LIN {X 0,Y 514.264,Z 1274.266,A -85,B 0,C 180,E1 4933.156,E2 4933.156} C_VEL
LIN {X 0,Y 513.464,Z 1291.981,A -85,B 0,C 180,E1 4937.266,E2 4937.266} C_VEL
LIN {X 0,Y 513.172,Z 1303.726,A -85,B 0,C 180,E1 4941.123,E2 4941.123} C_VEL
LIN {X 0,Y 512.967,Z 1310.956,A -85,B 0,C 180,E1 4944.936,E2 4944.936} C_VEL
LIN {X 0,Y 512.995,Z 1314.088,A -85,B 0,C 180,E1 4948.314,E2 4948.314} C_VEL
LIN {X 0,Y 513.103,Z 1314.089,A -85,B 0,C 180,E1 4951.685,E2 4951.685} C_VEL
LIN {X 0,Y 513.097,Z 1309.756,A -85,B 0,C 180,E1 4955.908,E2 4955.908} C_VEL
LIN {X 0,Y 513.202,Z 1300.306,A -85,B 0,C 180,E1 4960.161,E2 4960.161} C_VEL
LIN {X 0,Y 513.734,Z 1286.168,A -85,B 0,C 180,E1 4964.239,E2 4964.239} C_VEL
LIN {X 0,Y 514.771,Z 1266.36,A -85,B 0,C 180,E1 4968.328,E2 4968.328} C_VEL
LIN {X 0,Y 516.526,Z 1240.321,A -85,B 0,C 180,E1 4972.32,E2 4972.32} C_VEL
LIN {X 0,Y 518.823,Z 1209.462,A -85,B 0,C 180,E1 4975.866,E2 4975.866} C_VEL
LIN {X 0,Y 521.361,Z 1175.943,A -85,B 0,C 180,E1 4978.762,E2 4978.762} C_VEL
LIN {X 0,Y 523.842,Z 1140.515,A -85,B 0,C 180,E1 4981.019,E2 4981.019} C_VEL
LIN {X 0,Y 525.891,Z 1102.955,A -85,B 0,C 180,E1 4982.687,E2 4982.687} C_VEL
LIN {X 0,Y 527.428,Z 1065.762,A -85,B 0,C 180,E1 4983.695,E2 4983.695} C_VEL
LIN {X 0,Y 527.288,Z 1021.079,A -85,B 0,C 180,E1 4984.459,E2 4984.459} C_VEL
LIN {X 0,Y 512.361,Z 989.03,A -85,B 0,C 180,E1 4986.22,E2 4986.22} C_VEL
LIN {X 0,Y 512.298,Z 989.03,A -85,B 0,C 180,E1 4990.392,E2 4990.392} C_VEL
LIN {X 0,Y 512.249,Z 989.03,A -85,B 0,C 180,E1 4997.35,E2 4997.35} C_VEL
LIN {X 0,Y 512.299,Z 989.03,A -85,B 0,C 180,E1 5002.683,E2 5002.683} C_VEL
LIN {X 0,Y 512.294,Z 989.03,A -85,B 0,C 180,E1 5008.673,E2 5008.673} C_VEL
LIN {X 0,Y 512.37,Z 989.03,A -85,B 0,C 180,E1 5013.784,E2 5013.784} C_VEL
LIN {X 0,Y 512.546,Z 989.03,A -85,B 0,C 180,E1 5019.312,E2 5019.312} C_VEL
LIN {X 0,Y 512.454,Z 989.03,A -85,B 0,C 180,E1 5024.632,E2 5024.632} C_VEL
LIN {X 0,Y 512.627,Z 989.03,A -85,B 0,C 180,E1 5029.827,E2 5029.827} C_VEL
LIN {X 0,Y 512.838,Z 989.03,A -85,B 0,C 180,E1 5034.936,E2 5034.936} C_VEL
LIN {X 0,Y 512.854,Z 989.03,A -85,B 0,C 180,E1 5040,E2 5040} C_VEL
LIN {X 0,Y 512.807,Z 989.03,A -85,B 0,C 180,E1 5045.064,E2 5045.064} C_VEL
LIN {X 0,Y 512.702,Z 989.03,A -85,B 0,C 180,E1 5050.171,E2 5050.171} C_VEL
LIN {X 0,Y 512.597,Z 989.03,A -85,B 0,C 180,E1 5055.363,E2 5055.363} C_VEL
LIN {X 0,Y 512.537,Z 989.03,A -85,B 0,C 180,E1 5060.689,E2 5060.689} C_VEL
LIN {X 0,Y 512.336,Z 989.03,A -85,B 0,C 180,E1 5066.218,E2 5066.218} C_VEL
LIN {X 0,Y 512.295,Z 989.03,A -85,B 0,C 180,E1 5072.018,E2 5072.018} C_VEL
LIN {X 0,Y 512.168,Z 989.03,A -85,B 0,C 180,E1 5078.221,E2 5078.221} C_VEL
LIN {X 0,Y 512.21,Z 989.03,A -85,B 0,C 180,E1 5084.994,E2 5084.994} C_VEL
LIN {X 0,Y 512.302,Z 989.03,A -85,B 0,C 180,E1 5089.979,E2 5089.979} C_VEL
LIN {X 0,Y 512.239,Z 989.03,A -85,B 0,C 180,E1 5095.964,E2 5095.964} C_VEL
LIN {X 0,Y 512.363,Z 989.065,A -85,B 0,C 180,E1 5098.077,E2 5098.077} C_VEL
LIN {X 0,Y 521.604,Z 1021.148,A -85,B 0,C 180,E1 5100.836,E2 5100.836} C_VEL
LIN {X 0,Y 519.15,Z 1055.325,A -85,B 0,C 180,E1 5103.688,E2 5103.688} C_VEL
LIN {X 0,Y 516.857,Z 1085.604,A -85,B 0,C 180,E1 5107.034,E2 5107.034} C_VEL
LIN {X 0,Y 515.067,Z 1111.372,A -85,B 0,C 180,E1 5110.771,E2 5110.771} C_VEL
LIN {X 0,Y 513.907,Z 1131.701,A -85,B 0,C 180,E1 5114.677,E2 5114.677} C_VEL
LIN {X 0,Y 513.347,Z 1147.878,A -85,B 0,C 180,E1 5118.985,E2 5118.985} C_VEL
LIN {X 0,Y 513.104,Z 1158.306,A -85,B 0,C 180,E1 5123.245,E2 5123.245} C_VEL
LIN {X 0,Y 512.989,Z 1162.956,A -85,B 0,C 180,E1 5126.628,E2 5126.628} C_VEL
LIN {X 0,Y 513.004,Z 1164.497,A -85,B 0,C 180,E1 5130.001,E2 5130.001} C_VEL
LIN {X 0,Y 512.994,Z 1162.865,A -85,B 0,C 180,E1 5133.373,E2 5133.373} C_VEL
LIN {X 0,Y 513.065,Z 1156.495,A -85,B 0,C 180,E1 5137.606,E2 5137.606} C_VEL
LIN {X 0,Y 513.404,Z 1144.882,A -85,B 0,C 180,E1 5141.874,E2 5141.874} C_VEL
LIN {X 0,Y 514.188,Z 1127.29,A -85,B 0,C 180,E1 5146.189,E2 5146.189} C_VEL
LIN {X 0,Y 515.459,Z 1105.361,A -85,B 0,C 180,E1 5150.113,E2 5150.113} C_VEL
LIN {X 0,Y 517.484,Z 1077.478,A -85,B 0,C 180,E1 5153.867,E2 5153.867} C_VEL
LIN {X 0,Y 519.839,Z 1045.937,A -85,B 0,C 180,E1 5157.09,E2 5157.09} C_VEL
LIN {X 0,Y 521.275,Z 1018.437,A -85,B 0,C 180,E1 5159.305,E2 5159.305} C_VEL
LIN {X 0,Y 512.342,Z 989.03,A -85,B 0,C 180,E1 5161.88,E2 5161.88} C_VEL
LIN {X 0,Y 512.182,Z 989.03,A -85,B 0,C 180,E1 5168.223,E2 5168.223} C_VEL
LIN {X 0,Y 512.218,Z 989.03,A -85,B 0,C 180,E1 5175.007,E2 5175.007} C_VEL
LIN {X 0,Y 512.311,Z 989.03,A -85,B 0,C 180,E1 5179.982,E2 5179.982} C_VEL
LIN {X 0,Y 512.229,Z 989.03,A -85,B 0,C 180,E1 5185.964,E2 5185.964} C_VEL
LIN {X 0,Y 512.354,Z 989.03,A -85,B 0,C 180,E1 5192.078,E2 5192.078} C_VEL
LIN {X 0,Y 512.457,Z 989.03,A -85,B 0,C 180,E1 5197.494,E2 5197.494} C_VEL
LIN {X 0,Y 512.639,Z 989.03,A -85,B 0,C 180,E1 5202.882,E2 5202.882} C_VEL
LIN {X 0,Y 512.635,Z 989.03,A -85,B 0,C 180,E1 5209.828,E2 5209.828} C_VEL
LIN {X 0,Y 512.85,Z 989.03,A -85,B 0,C 180,E1 5214.936,E2 5214.936} C_VEL
LIN {X 0,Y 512.911,Z 989.03,A -85,B 0,C 180,E1 5220,E2 5220} C_VEL
LIN {X 0,Y 512.831,Z 989.03,A -85,B 0,C 180,E1 5225.064,E2 5225.064} C_VEL
LIN {X 0,Y 512.709,Z 989.03,A -85,B 0,C 180,E1 5230.171,E2 5230.171} C_VEL
LIN {X 0,Y 512.61,Z 989.03,A -85,B 0,C 180,E1 5235.363,E2 5235.363} C_VEL
LIN {X 0,Y 512.534,Z 989.03,A -85,B 0,C 180,E1 5240.689,E2 5240.689} C_VEL
LIN {X 0,Y 512.344,Z 989.03,A -85,B 0,C 180,E1 5246.217,E2 5246.217} C_VEL
LIN {X 0,Y 512.44,Z 989.03,A -85,B 0,C 180,E1 5252.008,E2 5252.008} C_VEL
LIN {X 0,Y 512.33,Z 989.03,A -85,B 0,C 180,E1 5258.061,E2 5258.061} C_VEL
LIN {X 0,Y 509.805,Z 989.03,A -85,B 0,C 180,E1 5259.49,E2 5259.49} C_VEL
LIN {X 0,Y 504.194,Z 989.03,A -85,B 0,C 180,E1 5261.878,E2 5261.878} C_VEL
LIN {X 0,Y 504.274,Z 989.03,A -85,B 0,C 180,E1 5268.424,E2 5268.424} C_VEL
LIN {X 0,Y 504.544,Z 989.315,A -85,B 0,C 180,E1 5273.26,E2 5273.26} C_VEL
LIN {X 0,Y 521.241,Z 1024.493,A -85,B 0,C 180,E1 5275.14,E2 5275.14} C_VEL
LIN {X 0,Y 520.227,Z 1081.386,A -85,B 0,C 180,E1 5276.169,E2 5276.169} C_VEL
LIN {X 0,Y 518.352,Z 1120.193,A -85,B 0,C 180,E1 5277.525,E2 5277.525} C_VEL
LIN {X 0,Y 515.742,Z 1157.972,A -85,B 0,C 180,E1 5279.553,E2 5279.553} C_VEL
LIN {X 0,Y 512.859,Z 1193.587,A -85,B 0,C 180,E1 5282.243,E2 5282.243} C_VEL
LIN {X 0,Y 510.276,Z 1224.521,A -85,B 0,C 180,E1 5285.369,E2 5285.369} C_VEL
LIN {X 0,Y 508.165,Z 1251.245,A -85,B 0,C 180,E1 5288.896,E2 5288.896} C_VEL
LIN {X 0,Y 506.553,Z 1274.264,A -85,B 0,C 180,E1 5292.891,E2 5292.891} C_VEL
LIN {X 0,Y 505.643,Z 1291.982,A -85,B 0,C 180,E1 5297.066,E2 5297.066} C_VEL
LIN {X 0,Y 505.264,Z 1304.676,A -85,B 0,C 180,E1 5301.411,E2 5301.411} C_VEL
LIN {X 0,Y 505.074,Z 1310.957,A -85,B 0,C 180,E1 5304.857,E2 5304.857} C_VEL
LIN {X 0,Y 505.093,Z 1314.088,A -85,B 0,C 180,E1 5308.287,E2 5308.287} C_VEL
LIN {X 0,Y 505.196,Z 1314.089,A -85,B 0,C 180,E1 5311.711,E2 5311.711} C_VEL
LIN {X 0,Y 505.205,Z 1309.756,A -85,B 0,C 180,E1 5316,E2 5316} C_VEL
LIN {X 0,Y 505.319,Z 1300.306,A -85,B 0,C 180,E1 5320.321,E2 5320.321} C_VEL
LIN {X 0,Y 505.986,Z 1285.076,A -85,B 0,C 180,E1 5324.738,E2 5324.738} C_VEL
LIN {X 0,Y 507.27,Z 1263.662,A -85,B 0,C 180,E1 5329.1,E2 5329.1} C_VEL
LIN {X 0,Y 509.094,Z 1238.474,A -85,B 0,C 180,E1 5332.912,E2 5332.912} C_VEL
LIN {X 0,Y 511.597,Z 1208.319,A -85,B 0,C 180,E1 5336.377,E2 5336.377} C_VEL
LIN {X 0,Y 514.358,Z 1175.174,A -85,B 0,C 180,E1 5339.252,E2 5339.252} C_VEL
LIN {X 0,Y 517.035,Z 1139.614,A -85,B 0,C 180,E1 5341.525,E2 5341.525} C_VEL
LIN {X 0,Y 519.276,Z 1101.697,A -85,B 0,C 180,E1 5343.205,E2 5343.205} C_VEL
LIN {X 0,Y 520.948,Z 1063.021,A -85,B 0,C 180,E1 5344.225,E2 5344.225} C_VEL
LIN {X 0,Y 520.741,Z 1023.716,A -85,B 0,C 180,E1 5344.911,E2 5344.911} C_VEL
LIN {X 0,Y 504.482,Z 989.03,A -85,B 0,C 180,E1 5346.818,E2 5346.818} C_VEL
LIN {X 0,Y 504.197,Z 989.03,A -85,B 0,C 180,E1 5353.5,E2 5353.5} C_VEL
LIN {X 0,Y 504.287,Z 989.03,A -85,B 0,C 180,E1 5358.83,E2 5358.83} C_VEL
LIN {X 0,Y 504.4,Z 989.03,A -85,B 0,C 180,E1 5363.876,E2 5363.876} C_VEL
LIN {X 0,Y 504.349,Z 989.03,A -85,B 0,C 180,E1 5370.189,E2 5370.189} C_VEL
LIN {X 0,Y 504.437,Z 989.03,A -85,B 0,C 180,E1 5375.242,E2 5375.242} C_VEL
LIN {X 0,Y 504.662,Z 989.03,A -85,B 0,C 180,E1 5380.798,E2 5380.798} C_VEL
LIN {X 0,Y 504.474,Z 989.03,A -85,B 0,C 180,E1 5386.155,E2 5386.155} C_VEL
LIN {X 0,Y 504.709,Z 989.03,A -85,B 0,C 180,E1 5391.403,E2 5391.403} C_VEL
LIN {X 0,Y 504.868,Z 989.03,A -85,B 0,C 180,E1 5396.573,E2 5396.573} C_VEL
LIN {X 0,Y 504.878,Z 989.03,A -85,B 0,C 180,E1 5401.713,E2 5401.713} C_VEL
LIN {X 0,Y 504.801,Z 989.03,A -85,B 0,C 180,E1 5406.867,E2 5406.867} C_VEL
LIN {X 0,Y 504.723,Z 989.03,A -85,B 0,C 180,E1 5412.08,E2 5412.08} C_VEL
LIN {X 0,Y 504.674,Z 989.03,A -85,B 0,C 180,E1 5417.397,E2 5417.397} C_VEL
LIN {X 0,Y 504.538,Z 989.03,A -85,B 0,C 180,E1 5422.88,E2 5422.88} C_VEL
LIN {X 0,Y 504.372,Z 989.03,A -85,B 0,C 180,E1 5428.599,E2 5428.599} C_VEL
LIN {X 0,Y 504.304,Z 989.03,A -85,B 0,C 180,E1 5434.646,E2 5434.646} C_VEL
LIN {X 0,Y 504.179,Z 989.03,A -85,B 0,C 180,E1 5441.18,E2 5441.18} C_VEL
LIN {X 0,Y 504.236,Z 989.03,A -85,B 0,C 180,E1 5446.504,E2 5446.504} C_VEL
LIN {X 0,Y 504.388,Z 989.03,A -85,B 0,C 180,E1 5453.249,E2 5453.249} C_VEL
LIN {X 0,Y 504.392,Z 989.133,A -85,B 0,C 180,E1 5457.512,E2 5457.512} C_VEL
LIN {X 0,Y 514.407,Z 1023.254,A -85,B 0,C 180,E1 5460.555,E2 5460.555} C_VEL
LIN {X 0,Y 511.797,Z 1056.465,A -85,B 0,C 180,E1 5463.398,E2 5463.398} C_VEL
LIN {X 0,Y 509.247,Z 1087.005,A -85,B 0,C 180,E1 5466.856,E2 5466.856} C_VEL
LIN {X 0,Y 507.312,Z 1112.759,A -85,B 0,C 180,E1 5470.702,E2 5470.702} C_VEL
LIN {X 0,Y 506.058,Z 1134.079,A -85,B 0,C 180,E1 5474.976,E2 5474.976} C_VEL
LIN {X 0,Y 505.494,Z 1150.423,A -85,B 0,C 180,E1 5479.682,E2 5479.682} C_VEL
LIN {X 0,Y 505.204,Z 1159.82,A -85,B 0,C 180,E1 5484,E2 5484} C_VEL
LIN {X 0,Y 505.088,Z 1164.116,A -85,B 0,C 180,E1 5488.289,E2 5488.289} C_VEL
LIN {X 0,Y 505.203,Z 1164.062,A -85,B 0,C 180,E1 5491.712,E2 5491.712} C_VEL
LIN {X 0,Y 505.158,Z 1159.685,A -85,B 0,C 180,E1 5496.002,E2 5496.002} C_VEL
LIN {X 0,Y 505.36,Z 1150.185,A -85,B 0,C 180,E1 5500.322,E2 5500.322} C_VEL
LIN {X 0,Y 505.989,Z 1134.907,A -85,B 0,C 180,E1 5504.736,E2 5504.736} C_VEL
LIN {X 0,Y 507.272,Z 1113.393,A -85,B 0,C 180,E1 5509.101,E2 5509.101} C_VEL
LIN {X 0,Y 509.165,Z 1088.092,A -85,B 0,C 180,E1 5512.914,E2 5512.914} C_VEL
LIN {X 0,Y 511.655,Z 1057.868,A -85,B 0,C 180,E1 5516.375,E2 5516.375} C_VEL
LIN {X 0,Y 514.45,Z 1024.571,A -85,B 0,C 180,E1 5519.249,E2 5519.249} C_VEL
LIN {X 0,Y 505.519,Z 992.998,A -85,B 0,C 180,E1 5522.083,E2 5522.083} C_VEL
LIN {X 0,Y 504.383,Z 989.03,A -85,B 0,C 180,E1 5522.459,E2 5522.459} C_VEL
LIN {X 0,Y 504.236,Z 989.03,A -85,B 0,C 180,E1 5528.937,E2 5528.937} C_VEL
LIN {X 0,Y 504.223,Z 989.03,A -85,B 0,C 180,E1 5534.092,E2 5534.092} C_VEL
LIN {X 0,Y 504.302,Z 989.03,A -85,B 0,C 180,E1 5538.832,E2 5538.832} C_VEL
LIN {X 0,Y 504.407,Z 989.03,A -85,B 0,C 180,E1 5543.877,E2 5543.877} C_VEL
LIN {X 0,Y 504.355,Z 989.03,A -85,B 0,C 180,E1 5550.19,E2 5550.19} C_VEL
LIN {X 0,Y 504.444,Z 989.03,A -85,B 0,C 180,E1 5555.242,E2 5555.242} C_VEL
LIN {X 0,Y 504.681,Z 989.03,A -85,B 0,C 180,E1 5560.799,E2 5560.799} C_VEL
LIN {X 0,Y 504.485,Z 989.03,A -85,B 0,C 180,E1 5566.156,E2 5566.156} C_VEL
LIN {X 0,Y 504.737,Z 989.03,A -85,B 0,C 180,E1 5571.403,E2 5571.403} C_VEL
LIN {X 0,Y 504.877,Z 989.03,A -85,B 0,C 180,E1 5576.573,E2 5576.573} C_VEL
LIN {X 0,Y 504.848,Z 989.03,A -85,B 0,C 180,E1 5581.713,E2 5581.713} C_VEL
LIN {X 0,Y 504.81,Z 989.03,A -85,B 0,C 180,E1 5586.867,E2 5586.867} C_VEL
LIN {X 0,Y 504.734,Z 989.03,A -85,B 0,C 180,E1 5592.08,E2 5592.08} C_VEL
LIN {X 0,Y 504.658,Z 989.03,A -85,B 0,C 180,E1 5597.398,E2 5597.398} C_VEL
LIN {X 0,Y 504.506,Z 989.03,A -85,B 0,C 180,E1 5602.881,E2 5602.881} C_VEL
LIN {X 0,Y 504.406,Z 989.03,A -85,B 0,C 180,E1 5608.597,E2 5608.597} C_VEL
LIN {X 0,Y 504.476,Z 989.03,A -85,B 0,C 180,E1 5614.633,E2 5614.633} C_VEL
LIN {X 0,Y 504.264,Z 989.03,A -85,B 0,C 180,E1 5621.172,E2 5621.172} C_VEL
LIN {X 0,Y 504.194,Z 989.03,A -85,B 0,C 180,E1 5621.878,E2 5621.878} C_VEL
LIN {X 0,Y 500.197,Z 989.03,A -85,B 0,C 180,E1 5623.826,E2 5623.826} C_VEL
LIN {X 0,Y 496.264,Z 989.03,A -85,B 0,C 180,E1 5625.804,E2 5625.804} C_VEL
LIN {X 0,Y 496.596,Z 989.03,A -85,B 0,C 180,E1 5632.573,E2 5632.573} C_VEL
LIN {X 0,Y 514.658,Z 1027.323,A -85,B 0,C 180,E1 5634.689,E2 5634.689} C_VEL
LIN {X 0,Y 513.661,Z 1081.286,A -85,B 0,C 180,E1 5635.675,E2 5635.675} C_VEL
LIN {X 0,Y 511.623,Z 1120.474,A -85,B 0,C 180,E1 5637.059,E2 5637.059} C_VEL
LIN {X 0,Y 508.83,Z 1157.545,A -85,B 0,C 180,E1 5639.064,E2 5639.064} C_VEL
LIN {X 0,Y 505.715,Z 1193.156,A -85,B 0,C 180,E1 5641.775,E2 5641.775} C_VEL
LIN {X 0,Y 502.879,Z 1224.715,A -85,B 0,C 180,E1 5645.006,E2 5645.006} C_VEL
LIN {X 0,Y 500.454,Z 1252.697,A -85,B 0,C 180,E1 5648.786,E2 5648.786} C_VEL
LIN {X 0,Y 498.725,Z 1275.344,A -85,B 0,C 180,E1 5652.841,E2 5652.841} C_VEL
LIN {X 0,Y 497.812,Z 1291.982,A -85,B 0,C 180,E1 5656.858,E2 5656.858} C_VEL
LIN {X 0,Y 497.388,Z 1304.676,A -85,B 0,C 180,E1 5661.274,E2 5661.274} C_VEL
LIN {X 0,Y 497.182,Z 1310.957,A -85,B 0,C 180,E1 5664.775,E2 5664.775} C_VEL
LIN {X 0,Y 497.214,Z 1314.088,A -85,B 0,C 180,E1 5668.26,E2 5668.26} C_VEL
LIN {X 0,Y 497.291,Z 1314.089,A -85,B 0,C 180,E1 5671.738,E2 5671.738} C_VEL
LIN {X 0,Y 497.327,Z 1309.755,A -85,B 0,C 180,E1 5676.096,E2 5676.096} C_VEL
LIN {X 0,Y 497.438,Z 1300.306,A -85,B 0,C 180,E1 5680.486,E2 5680.486} C_VEL
LIN {X 0,Y 498.235,Z 1284.679,A -85,B 0,C 180,E1 5685.075,E2 5685.075} C_VEL
LIN {X 0,Y 499.604,Z 1263.661,A -85,B 0,C 180,E1 5689.404,E2 5689.404} C_VEL
LIN {X 0,Y 501.633,Z 1238.473,A -85,B 0,C 180,E1 5693.273,E2 5693.273} C_VEL
LIN {X 0,Y 504.345,Z 1208.416,A -85,B 0,C 180,E1 5696.776,E2 5696.776} C_VEL
LIN {X 0,Y 507.368,Z 1174.406,A -85,B 0,C 180,E1 5699.756,E2 5699.756} C_VEL
LIN {X 0,Y 510.363,Z 1137.859,A -85,B 0,C 180,E1 5702.089,E2 5702.089} C_VEL
LIN {X 0,Y 512.762,Z 1099.707,A -85,B 0,C 180,E1 5703.759,E2 5703.759} C_VEL
LIN {X 0,Y 514.393,Z 1061.693,A -85,B 0,C 180,E1 5704.742,E2 5704.742} C_VEL
LIN {X 0,Y 514.105,Z 1026.127,A -85,B 0,C 180,E1 5705.372,E2 5705.372} C_VEL
LIN {X 0,Y 496.553,Z 989.03,A -85,B 0,C 180,E1 5707.429,E2 5707.429} C_VEL
LIN {X 0,Y 496.322,Z 989.03,A -85,B 0,C 180,E1 5714.369,E2 5714.369} C_VEL
LIN {X 0,Y 496.387,Z 989.03,A -85,B 0,C 180,E1 5720.33,E2 5720.33} C_VEL
LIN {X 0,Y 496.374,Z 989.03,A -85,B 0,C 180,E1 5726.826,E2 5726.826} C_VEL
LIN {X 0,Y 496.475,Z 989.03,A -85,B 0,C 180,E1 5732.877,E2 5732.877} C_VEL
LIN {X 0,Y 496.659,Z 989.03,A -85,B 0,C 180,E1 5738.618,E2 5738.618} C_VEL
LIN {X 0,Y 496.666,Z 989.03,A -85,B 0,C 180,E1 5744.131,E2 5744.131} C_VEL
LIN {X 0,Y 496.773,Z 989.03,A -85,B 0,C 180,E1 5749.499,E2 5749.499} C_VEL
LIN {X 0,Y 497.027,Z 989.03,A -85,B 0,C 180,E1 5754.774,E2 5754.774} C_VEL
LIN {X 0,Y 497.061,Z 989.03,A -85,B 0,C 180,E1 5760,E2 5760} C_VEL
LIN {X 0,Y 496.993,Z 989.03,A -85,B 0,C 180,E1 5765.226,E2 5765.226} C_VEL
LIN {X 0,Y 496.864,Z 989.03,A -85,B 0,C 180,E1 5770.499,E2 5770.499} C_VEL
LIN {X 0,Y 496.754,Z 989.03,A -85,B 0,C 180,E1 5775.866,E2 5775.866} C_VEL
LIN {X 0,Y 496.656,Z 989.03,A -85,B 0,C 180,E1 5781.382,E2 5781.382} C_VEL
LIN {X 0,Y 496.454,Z 989.03,A -85,B 0,C 180,E1 5787.124,E2 5787.124} C_VEL
LIN {X 0,Y 496.392,Z 989.03,A -85,B 0,C 180,E1 5793.173,E2 5793.173} C_VEL
LIN {X 0,Y 496.228,Z 989.03,A -85,B 0,C 180,E1 5799.685,E2 5799.685} C_VEL
LIN {X 0,Y 496.335,Z 989.03,A -85,B 0,C 180,E1 5805.632,E2 5805.632} C_VEL
LIN {X 0,Y 496.417,Z 989.03,A -85,B 0,C 180,E1 5812.215,E2 5812.215} C_VEL
LIN {X 0,Y 496.429,Z 989.297,A -85,B 0,C 180,E1 5816.829,E2 5816.829} C_VEL
LIN {X 0,Y 507.224,Z 1025.443,A -85,B 0,C 180,E1 5820.272,E2 5820.272} C_VEL
LIN {X 0,Y 504.259,Z 1059.901,A -85,B 0,C 180,E1 5823.329,E2 5823.329} C_VEL
LIN {X 0,Y 501.447,Z 1090.626,A -85,B 0,C 180,E1 5826.971,E2 5826.971} C_VEL
LIN {X 0,Y 499.442,Z 1116.379,A -85,B 0,C 180,E1 5831.047,E2 5831.047} C_VEL
LIN {X 0,Y 498.188,Z 1135.456,A -85,B 0,C 180,E1 5835.079,E2 5835.079} C_VEL
LIN {X 0,Y 497.608,Z 1150.422,A -85,B 0,C 180,E1 5839.517,E2 5839.517} C_VEL
LIN {X 0,Y 497.33,Z 1159.819,A -85,B 0,C 180,E1 5843.904,E2 5843.904} C_VEL
LIN {X 0,Y 497.21,Z 1164.116,A -85,B 0,C 180,E1 5848.261,E2 5848.261} C_VEL
LIN {X 0,Y 497.297,Z 1164.063,A -85,B 0,C 180,E1 5851.739,E2 5851.739} C_VEL
LIN {X 0,Y 497.251,Z 1159.686,A -85,B 0,C 180,E1 5856.098,E2 5856.098} C_VEL
LIN {X 0,Y 497.463,Z 1150.187,A -85,B 0,C 180,E1 5860.487,E2 5860.487} C_VEL
LIN {X 0,Y 498.186,Z 1135.116,A -85,B 0,C 180,E1 5864.92,E2 5864.92} C_VEL
LIN {X 0,Y 499.496,Z 1114.688,A -85,B 0,C 180,E1 5869.181,E2 5869.181} C_VEL
LIN {X 0,Y 501.647,Z 1088.097,A -85,B 0,C 180,E1 5873.278,E2 5873.278} C_VEL
LIN {X 0,Y 504.376,Z 1057.964,A -85,B 0,C 180,E1 5876.776,E2 5876.776} C_VEL
LIN {X 0,Y 507.268,Z 1024.909,A -85,B 0,C 180,E1 5879.678,E2 5879.678} C_VEL
LIN {X 0,Y 496.419,Z 989.03,A -85,B 0,C 180,E1 5883.173,E2 5883.173} C_VEL
LIN {X 0,Y 496.232,Z 989.03,A -85,B 0,C 180,E1 5889.688,E2 5889.688} C_VEL
LIN {X 0,Y 496.342,Z 989.03,A -85,B 0,C 180,E1 5895.635,E2 5895.635} C_VEL
LIN {X 0,Y 496.428,Z 989.03,A -85,B 0,C 180,E1 5902.218,E2 5902.218} C_VEL
LIN {X 0,Y 496.352,Z 989.03,A -85,B 0,C 180,E1 5908.35,E2 5908.35} C_VEL
LIN {X 0,Y 496.538,Z 989.03,A -85,B 0,C 180,E1 5914.821,E2 5914.821} C_VEL
LIN {X 0,Y 496.732,Z 989.03,A -85,B 0,C 180,E1 5920.479,E2 5920.479} C_VEL
LIN {X 0,Y 496.597,Z 989.03,A -85,B 0,C 180,E1 5926.507,E2 5926.507} C_VEL
LIN {X 0,Y 497.006,Z 989.03,A -85,B 0,C 180,E1 5933.025,E2 5933.025} C_VEL
LIN {X 0,Y 497.238,Z 989.03,A -85,B 0,C 180,E1 5938.261,E2 5938.261} C_VEL
LIN {X 0,Y 497.014,Z 989.03,A -85,B 0,C 180,E1 5945.226,E2 5945.226} C_VEL
LIN {X 0,Y 496.872,Z 989.03,A -85,B 0,C 180,E1 5950.499,E2 5950.499} C_VEL
LIN {X 0,Y 496.756,Z 989.03,A -85,B 0,C 180,E1 5955.866,E2 5955.866} C_VEL
LIN {X 0,Y 496.655,Z 989.03,A -85,B 0,C 180,E1 5961.382,E2 5961.382} C_VEL
LIN {X 0,Y 496.474,Z 989.03,A -85,B 0,C 180,E1 5967.123,E2 5967.123} C_VEL
LIN {X 0,Y 496.546,Z 989.03,A -85,B 0,C 180,E1 5973.161,E2 5973.161} C_VEL
LIN {X 0,Y 496.385,Z 989.03,A -85,B 0,C 180,E1 5979.671,E2 5979.671} C_VEL
LIN {X 0,Y 496.264,Z 989.03,A -85,B 0,C 180,E1 5985.804,E2 5985.804} C_VEL
LIN {X 0,Y 492.339,Z 989.03,A -85,B 0,C 180,E1 5987.779,E2 5987.779} C_VEL
LIN {X 0,Y 488.455,Z 989.03,A -85,B 0,C 180,E1 5989.785,E2 5989.785} C_VEL
LIN {X 0,Y 488.649,Z 989.274,A -85,B 0,C 180,E1 5991.919,E2 5991.919} C_VEL
LIN {X 0,Y 508.023,Z 1028.77,A -85,B 0,C 180,E1 5994.206,E2 5994.206} C_VEL
LIN {X 0,Y 506.923,Z 1081.953,A -85,B 0,C 180,E1 5995.22,E2 5995.22} C_VEL
LIN {X 0,Y 504.79,Z 1121.445,A -85,B 0,C 180,E1 5996.629,E2 5996.629} C_VEL
LIN {X 0,Y 501.901,Z 1157.667,A -85,B 0,C 180,E1 5998.598,E2 5998.598} C_VEL
LIN {X 0,Y 498.58,Z 1193.456,A -85,B 0,C 180,E1 6001.364,E2 6001.364} C_VEL
LIN {X 0,Y 495.49,Z 1224.906,A -85,B 0,C 180,E1 6004.632,E2 6004.632} C_VEL
LIN {X 0,Y 492.896,Z 1252.695,A -85,B 0,C 180,E1 6008.445,E2 6008.445} C_VEL
LIN {X 0,Y 491.137,Z 1273.884,A -85,B 0,C 180,E1 6012.256,E2 6012.256} C_VEL
LIN {X 0,Y 490.012,Z 1291.981,A -85,B 0,C 180,E1 6016.645,E2 6016.645} C_VEL
LIN {X 0,Y 489.507,Z 1304.676,A -85,B 0,C 180,E1 6021.133,E2 6021.133} C_VEL
LIN {X 0,Y 489.292,Z 1310.956,A -85,B 0,C 180,E1 6024.691,E2 6024.691} C_VEL
LIN {X 0,Y 489.311,Z 1314.088,A -85,B 0,C 180,E1 6028.232,E2 6028.232} C_VEL
LIN {X 0,Y 489.385,Z 1314.089,A -85,B 0,C 180,E1 6031.766,E2 6031.766} C_VEL
LIN {X 0,Y 489.432,Z 1309.755,A -85,B 0,C 180,E1 6036.194,E2 6036.194} C_VEL
LIN {X 0,Y 489.574,Z 1300.307,A -85,B 0,C 180,E1 6040.657,E2 6040.657} C_VEL
LIN {X 0,Y 490.392,Z 1285.291,A -85,B 0,C 180,E1 6045.162,E2 6045.162} C_VEL
LIN {X 0,Y 491.954,Z 1263.659,A -85,B 0,C 180,E1 6049.719,E2 6049.719} C_VEL
LIN {X 0,Y 494.271,Z 1237.429,A -85,B 0,C 180,E1 6053.783,E2 6053.783} C_VEL
LIN {X 0,Y 497.199,Z 1207.529,A -85,B 0,C 180,E1 6057.286,E2 6057.286} C_VEL
LIN {X 0,Y 500.392,Z 1174.402,A -85,B 0,C 180,E1 6060.214,E2 6060.214} C_VEL
LIN {X 0,Y 503.524,Z 1138.858,A -85,B 0,C 180,E1 6062.518,E2 6062.518} C_VEL
LIN {X 0,Y 506.006,Z 1099.903,A -85,B 0,C 180,E1 6064.223,E2 6064.223} C_VEL
LIN {X 0,Y 507.842,Z 1060.043,A -85,B 0,C 180,E1 6065.261,E2 6065.261} C_VEL
LIN {X 0,Y 507.59,Z 1028.789,A -85,B 0,C 180,E1 6065.828,E2 6065.828} C_VEL
LIN {X 0,Y 488.605,Z 989.03,A -85,B 0,C 180,E1 6068.146,E2 6068.146} C_VEL
LIN {X 0,Y 488.41,Z 989.03,A -85,B 0,C 180,E1 6074.717,E2 6074.717} C_VEL
LIN {X 0,Y 488.463,Z 989.03,A -85,B 0,C 180,E1 6080.562,E2 6080.562} C_VEL
LIN {X 0,Y 488.466,Z 989.03,A -85,B 0,C 180,E1 6086.522,E2 6086.522} C_VEL
LIN {X 0,Y 488.546,Z 989.03,A -85,B 0,C 180,E1 6092.4,E2 6092.4} C_VEL
LIN {X 0,Y 488.694,Z 989.03,A -85,B 0,C 180,E1 6098.252,E2 6098.252} C_VEL
LIN {X 0,Y 488.75,Z 989.03,A -85,B 0,C 180,E1 6103.867,E2 6103.867} C_VEL
LIN {X 0,Y 488.85,Z 989.03,A -85,B 0,C 180,E1 6109.327,E2 6109.327} C_VEL
LIN {X 0,Y 489.114,Z 989.03,A -85,B 0,C 180,E1 6114.69,E2 6114.69} C_VEL
LIN {X 0,Y 489.16,Z 989.03,A -85,B 0,C 180,E1 6120,E2 6120} C_VEL
LIN {X 0,Y 489.078,Z 989.03,A -85,B 0,C 180,E1 6125.311,E2 6125.311} C_VEL
LIN {X 0,Y 488.937,Z 989.03,A -85,B 0,C 180,E1 6130.671,E2 6130.671} C_VEL
LIN {X 0,Y 488.784,Z 989.03,A -85,B 0,C 180,E1 6136.854,E2 6136.854} C_VEL
LIN {X 0,Y 488.687,Z 989.03,A -85,B 0,C 180,E1 6142.126,E2 6142.126} C_VEL
LIN {X 0,Y 488.53,Z 989.03,A -85,B 0,C 180,E1 6147.601,E2 6147.601} C_VEL
LIN {X 0,Y 488.456,Z 989.03,A -85,B 0,C 180,E1 6153.784,E2 6153.784} C_VEL
LIN {X 0,Y 488.332,Z 989.03,A -85,B 0,C 180,E1 6160.459,E2 6160.459} C_VEL
LIN {X 0,Y 488.413,Z 989.03,A -85,B 0,C 180,E1 6165.282,E2 6165.282} C_VEL
LIN {X 0,Y 488.489,Z 989.03,A -85,B 0,C 180,E1 6171.843,E2 6171.843} C_VEL
LIN {X 0,Y 488.505,Z 989.404,A -85,B 0,C 180,E1 6176.117,E2 6176.117} C_VEL
LIN {X 0,Y 498.448,Z 1021.358,A -85,B 0,C 180,E1 6179.361,E2 6179.361} C_VEL
LIN {X 0,Y 499.885,Z 1029.479,A -85,B 0,C 180,E1 6180.124,E2 6180.124} C_VEL
LIN {X 0,Y 496.61,Z 1063.94,A -85,B 0,C 180,E1 6183.342,E2 6183.342} C_VEL
LIN {X 0,Y 493.792,Z 1092.223,A -85,B 0,C 180,E1 6186.831,E2 6186.831} C_VEL
LIN {X 0,Y 491.805,Z 1116.374,A -85,B 0,C 180,E1 6190.741,E2 6190.741} C_VEL
LIN {X 0,Y 490.365,Z 1135.462,A -85,B 0,C 180,E1 6194.837,E2 6194.837} C_VEL
LIN {X 0,Y 489.734,Z 1150.42,A -85,B 0,C 180,E1 6199.347,E2 6199.347} C_VEL
LIN {X 0,Y 489.439,Z 1159.817,A -85,B 0,C 180,E1 6203.806,E2 6203.806} C_VEL
LIN {X 0,Y 489.306,Z 1164.116,A -85,B 0,C 180,E1 6208.233,E2 6208.233} C_VEL
LIN {X 0,Y 489.391,Z 1164.063,A -85,B 0,C 180,E1 6211.768,E2 6211.768} C_VEL
LIN {X 0,Y 489.342,Z 1159.687,A -85,B 0,C 180,E1 6216.197,E2 6216.197} C_VEL
LIN {X 0,Y 489.584,Z 1150.189,A -85,B 0,C 180,E1 6220.658,E2 6220.658} C_VEL
LIN {X 0,Y 490.389,Z 1135.116,A -85,B 0,C 180,E1 6225.163,E2 6225.163} C_VEL
LIN {X 0,Y 491.904,Z 1113.399,A -85,B 0,C 180,E1 6229.722,E2 6229.722} C_VEL
LIN {X 0,Y 494.305,Z 1087.084,A -85,B 0,C 180,E1 6233.784,E2 6233.784} C_VEL
LIN {X 0,Y 497.269,Z 1057.07,A -85,B 0,C 180,E1 6237.286,E2 6237.286} C_VEL
LIN {X 0,Y 499.947,Z 1026.887,A -85,B 0,C 180,E1 6239.997,E2 6239.997} C_VEL
LIN {X 0,Y 490.111,Z 993.78,A -85,B 0,C 180,E1 6243.358,E2 6243.358} C_VEL
LIN {X 0,Y 488.467,Z 989.03,A -85,B 0,C 180,E1 6243.887,E2 6243.887} C_VEL
LIN {X 0,Y 488.334,Z 989.03,A -85,B 0,C 180,E1 6250.462,E2 6250.462} C_VEL
LIN {X 0,Y 488.42,Z 989.03,A -85,B 0,C 180,E1 6255.285,E2 6255.285} C_VEL
LIN {X 0,Y 488.5,Z 989.03,A -85,B 0,C 180,E1 6261.845,E2 6261.845} C_VEL
LIN {X 0,Y 488.449,Z 989.03,A -85,B 0,C 180,E1 6268.32,E2 6268.32} C_VEL
LIN {X 0,Y 488.574,Z 989.03,A -85,B 0,C 180,E1 6274.381,E2 6274.381} C_VEL
LIN {X 0,Y 488.81,Z 989.03,A -85,B 0,C 180,E1 6280.15,E2 6280.15} C_VEL
LIN {X 0,Y 488.663,Z 989.03,A -85,B 0,C 180,E1 6285.698,E2 6285.698} C_VEL
LIN {X 0,Y 488.923,Z 989.03,A -85,B 0,C 180,E1 6291.123,E2 6291.123} C_VEL
LIN {X 0,Y 489.087,Z 989.03,A -85,B 0,C 180,E1 6296.462,E2 6296.462} C_VEL
LIN {X 0,Y 489.07,Z 989.03,A -85,B 0,C 180,E1 6301.768,E2 6301.768} C_VEL
LIN {X 0,Y 489.01,Z 989.03,A -85,B 0,C 180,E1 6307.09,E2 6307.09} C_VEL
LIN {X 0,Y 488.939,Z 989.03,A -85,B 0,C 180,E1 6312.476,E2 6312.476} C_VEL
LIN {X 0,Y 488.78,Z 989.03,A -85,B 0,C 180,E1 6317.982,E2 6317.982} C_VEL
LIN {X 0,Y 488.645,Z 989.03,A -85,B 0,C 180,E1 6323.668,E2 6323.668} C_VEL
LIN {X 0,Y 488.518,Z 989.03,A -85,B 0,C 180,E1 6330.126,E2 6330.126} C_VEL
LIN {X 0,Y 488.552,Z 989.03,A -85,B 0,C 180,E1 6335.933,E2 6335.933} C_VEL
LIN {X 0,Y 488.386,Z 989.03,A -85,B 0,C 180,E1 6342.135,E2 6342.135} C_VEL
LIN {X 0,Y 488.409,Z 989.03,A -85,B 0,C 180,E1 6347.858,E2 6347.858} C_VEL
LIN {X 0,Y 488.455,Z 989.03,A -85,B 0,C 180,E1 6349.785,E2 6349.785} C_VEL
LIN {X 0,Y 488.27,Z 992.282,A -85,B 0,C 180,E1 6350.825,E2 6350.825} C_VEL
LIN {X 0,Y 488.847,Z 1003.07,A -85,B 0,C 180,E1 6351.958,E2 6351.958} C_VEL
LIN {X 0,Y 492.058,Z 1012.441,A -85,B 0,C 180,E1 6352.627,E2 6352.627} C_VEL
LIN {X 0,Y 501.578,Z 1032.893,A -85,B 0,C 180,E1 6353.768,E2 6353.768} C_VEL
LIN {X 0,Y 500.223,Z 1082.335,A -85,B 0,C 180,E1 6354.745,E2 6354.745} C_VEL
LIN {X 0,Y 497.935,Z 1120.184,A -85,B 0,C 180,E1 6356.118,E2 6356.118} C_VEL
LIN {X 0,Y 494.78,Z 1159.31,A -85,B 0,C 180,E1 6358.257,E2 6358.257} C_VEL
LIN {X 0,Y 491.635,Z 1192.198,A -85,B 0,C 180,E1 6360.795,E2 6360.795} C_VEL
LIN {X 0,Y 488.238,Z 1224.284,A -85,B 0,C 180,E1 6364.147,E2 6364.147} C_VEL
LIN {X 0,Y 485.519,Z 1251.24,A -85,B 0,C 180,E1 6367.861,E2 6367.861} C_VEL
LIN {X 0,Y 483.353,Z 1274.585,A -85,B 0,C 180,E1 6372.114,E2 6372.114} C_VEL
LIN {X 0,Y 482.146,Z 1292.615,A -85,B 0,C 180,E1 6376.615,E2 6376.615} C_VEL
LIN {X 0,Y 481.649,Z 1304.677,A -85,B 0,C 180,E1 6380.987,E2 6380.987} C_VEL
LIN {X 0,Y 481.401,Z 1310.956,A -85,B 0,C 180,E1 6384.603,E2 6384.603} C_VEL
LIN {X 0,Y 481.423,Z 1314.088,A -85,B 0,C 180,E1 6388.203,E2 6388.203} C_VEL
LIN {X 0,Y 481.484,Z 1314.09,A -85,B 0,C 180,E1 6391.795,E2 6391.795} C_VEL
LIN {X 0,Y 481.548,Z 1309.755,A -85,B 0,C 180,E1 6396.296,E2 6396.296} C_VEL
LIN {X 0,Y 481.713,Z 1300.307,A -85,B 0,C 180,E1 6400.833,E2 6400.833} C_VEL
LIN {X 0,Y 482.61,Z 1285.291,A -85,B 0,C 180,E1 6405.412,E2 6405.412} C_VEL
LIN {X 0,Y 484.324,Z 1263.658,A -85,B 0,C 180,E1 6410.042,E2 6410.042} C_VEL
LIN {X 0,Y 486.846,Z 1237.165,A -85,B 0,C 180,E1 6414.205,E2 6414.205} C_VEL
LIN {X 0,Y 489.971,Z 1207.782,A -85,B 0,C 180,E1 6417.696,E2 6417.696} C_VEL
LIN {X 0,Y 493.438,Z 1174.49,A -85,B 0,C 180,E1 6420.677,E2 6420.677} C_VEL
LIN {X 0,Y 496.594,Z 1137.525,A -85,B 0,C 180,E1 6423.029,E2 6423.029} C_VEL
LIN {X 0,Y 499.346,Z 1097.64,A -85,B 0,C 180,E1 6424.777,E2 6424.777} C_VEL
LIN {X 0,Y 501.37,Z 1056.812,A -85,B 0,C 180,E1 6425.823,E2 6425.823} C_VEL
LIN {X 0,Y 501.273,Z 1031.759,A -85,B 0,C 180,E1 6426.276,E2 6426.276} C_VEL
LIN {X 0,Y 480.62,Z 989.03,A -85,B 0,C 180,E1 6428.898,E2 6428.898} C_VEL
LIN {X 0,Y 480.444,Z 989.03,A -85,B 0,C 180,E1 6433.75,E2 6433.75} C_VEL
LIN {X 0,Y 480.508,Z 989.03,A -85,B 0,C 180,E1 6438.912,E2 6438.912} C_VEL
LIN {X 0,Y 480.498,Z 989.03,A -85,B 0,C 180,E1 6444.738,E2 6444.738} C_VEL
LIN {X 0,Y 480.54,Z 989.03,A -85,B 0,C 180,E1 6449.84,E2 6449.84} C_VEL
LIN {X 0,Y 480.681,Z 989.03,A -85,B 0,C 180,E1 6455.915,E2 6455.915} C_VEL
LIN {X 0,Y 480.89,Z 989.03,A -85,B 0,C 180,E1 6461.713,E2 6461.713} C_VEL
LIN {X 0,Y 480.798,Z 989.03,A -85,B 0,C 180,E1 6467.309,E2 6467.309} C_VEL
LIN {X 0,Y 481.147,Z 989.03,A -85,B 0,C 180,E1 6472.793,E2 6472.793} C_VEL
LIN {X 0,Y 481.422,Z 989.03,A -85,B 0,C 180,E1 6478.204,E2 6478.204} C_VEL
LIN {X 0,Y 481.299,Z 989.03,A -85,B 0,C 180,E1 6483.595,E2 6483.595} C_VEL
LIN {X 0,Y 481.093,Z 989.03,A -85,B 0,C 180,E1 6489.023,E2 6489.023} C_VEL
LIN {X 0,Y 480.974,Z 989.03,A -85,B 0,C 180,E1 6494.536,E2 6494.536} C_VEL
LIN {X 0,Y 480.83,Z 989.03,A -85,B 0,C 180,E1 6500.194,E2 6500.194} C_VEL
LIN {X 0,Y 480.656,Z 989.03,A -85,B 0,C 180,E1 6506.072,E2 6506.072} C_VEL
LIN {X 0,Y 480.522,Z 989.03,A -85,B 0,C 180,E1 6512.265,E2 6512.265} C_VEL
LIN {X 0,Y 480.398,Z 989.03,A -85,B 0,C 180,E1 6518.918,E2 6518.918} C_VEL
LIN {X 0,Y 480.416,Z 989.03,A -85,B 0,C 180,E1 6523.744,E2 6523.744} C_VEL
LIN {X 0,Y 480.487,Z 989.03,A -85,B 0,C 180,E1 6528.913,E2 6528.913} C_VEL
LIN {X 0,Y 480.588,Z 989.03,A -85,B 0,C 180,E1 6535.157,E2 6535.157} C_VEL
LIN {X 0,Y 480.808,Z 990.837,A -85,B 0,C 180,E1 6535.486,E2 6535.486} C_VEL
LIN {X 0,Y 489.079,Z 1014.658,A -85,B 0,C 180,E1 6538.015,E2 6538.015} C_VEL
LIN {X 0,Y 492.718,Z 1031.175,A -85,B 0,C 180,E1 6539.793,E2 6539.793} C_VEL
LIN {X 0,Y 489.303,Z 1064.27,A -85,B 0,C 180,E1 6542.952,E2 6542.952} C_VEL
LIN {X 0,Y 486.34,Z 1092.216,A -85,B 0,C 180,E1 6546.455,E2 6546.455} C_VEL
LIN {X 0,Y 484.07,Z 1116.369,A -85,B 0,C 180,E1 6550.421,E2 6550.421} C_VEL
LIN {X 0,Y 482.556,Z 1135.46,A -85,B 0,C 180,E1 6554.586,E2 6554.586} C_VEL
LIN {X 0,Y 481.844,Z 1150.418,A -85,B 0,C 180,E1 6559.17,E2 6559.17} C_VEL
LIN {X 0,Y 481.556,Z 1159.816,A -85,B 0,C 180,E1 6563.704,E2 6563.704} C_VEL
LIN {X 0,Y 481.418,Z 1164.116,A -85,B 0,C 180,E1 6568.204,E2 6568.204} C_VEL
LIN {X 0,Y 481.49,Z 1164.064,A -85,B 0,C 180,E1 6571.797,E2 6571.797} C_VEL
LIN {X 0,Y 481.466,Z 1159.688,A -85,B 0,C 180,E1 6576.298,E2 6576.298} C_VEL
LIN {X 0,Y 481.717,Z 1150.191,A -85,B 0,C 180,E1 6580.834,E2 6580.834} C_VEL
LIN {X 0,Y 482.604,Z 1135.12,A -85,B 0,C 180,E1 6585.414,E2 6585.414} C_VEL
LIN {X 0,Y 484.269,Z 1113.402,A -85,B 0,C 180,E1 6590.046,E2 6590.046} C_VEL
LIN {X 0,Y 486.938,Z 1086.842,A -85,B 0,C 180,E1 6594.201,E2 6594.201} C_VEL
LIN {X 0,Y 490.049,Z 1057.333,A -85,B 0,C 180,E1 6597.695,E2 6597.695} C_VEL
LIN {X 0,Y 492.819,Z 1029.486,A -85,B 0,C 180,E1 6600.274,E2 6600.274} C_VEL
LIN {X 0,Y 484.132,Z 999.035,A -85,B 0,C 180,E1 6603.555,E2 6603.555} C_VEL
LIN {X 0,Y 480.605,Z 989.03,A -85,B 0,C 180,E1 6604.625,E2 6604.625} C_VEL
LIN {X 0,Y 480.407,Z 989.03,A -85,B 0,C 180,E1 6611.273,E2 6611.273} C_VEL
LIN {X 0,Y 480.452,Z 989.03,A -85,B 0,C 180,E1 6616.295,E2 6616.295} C_VEL
LIN {X 0,Y 480.607,Z 989.03,A -85,B 0,C 180,E1 6621.717,E2 6621.717} C_VEL
LIN {X 0,Y 480.537,Z 989.03,A -85,B 0,C 180,E1 6627.982,E2 6627.982} C_VEL
LIN {X 0,Y 480.664,Z 989.03,A -85,B 0,C 180,E1 6633.928,E2 6633.928} C_VEL
LIN {X 0,Y 480.896,Z 989.03,A -85,B 0,C 180,E1 6640.286,E2 6640.286} C_VEL
LIN {X 0,Y 480.751,Z 989.03,A -85,B 0,C 180,E1 6645.458,E2 6645.458} C_VEL
LIN {X 0,Y 481.04,Z 989.03,A -85,B 0,C 180,E1 6650.976,E2 6650.976} C_VEL
LIN {X 0,Y 481.21,Z 989.03,A -85,B 0,C 180,E1 6656.404,E2 6656.404} C_VEL
LIN {X 0,Y 481.194,Z 989.03,A -85,B 0,C 180,E1 6661.797,E2 6661.797} C_VEL
LIN {X 0,Y 481.095,Z 989.03,A -85,B 0,C 180,E1 6667.207,E2 6667.207} C_VEL
LIN {X 0,Y 480.974,Z 989.03,A -85,B 0,C 180,E1 6673.441,E2 6673.441} C_VEL
LIN {X 0,Y 480.851,Z 989.03,A -85,B 0,C 180,E1 6679.699,E2 6679.699} C_VEL
LIN {X 0,Y 480.655,Z 989.03,A -85,B 0,C 180,E1 6686.073,E2 6686.073} C_VEL
LIN {X 0,Y 480.656,Z 989.03,A -85,B 0,C 180,E1 6692.255,E2 6692.255} C_VEL
LIN {X 0,Y 480.58,Z 989.03,A -85,B 0,C 180,E1 6698.9,E2 6698.9} C_VEL
LIN {X 0,Y 480.401,Z 989.03,A -85,B 0,C 180,E1 6703.741,E2 6703.741} C_VEL
LIN {X 0,Y 480.479,Z 989.03,A -85,B 0,C 180,E1 6709.788,E2 6709.788} C_VEL
LIN {X 0,Y 480.659,Z 989.237,A -85,B 0,C 180,E1 6711.201,E2 6711.201} C_VEL
LIN {X 0,Y 492.058,Z 1012.441,A -85,B 0,C 180,E1 6712.627,E2 6712.627} C_VEL
LIN {X 0,Y 495.195,Z 1022.185,A -85,B 0,C 180,E1 6713.062,E2 6713.062} C_VEL
LIN {X 0,Y 494.951,Z 1046.987,A -85,B 0,C 180,E1 6713.475,E2 6713.475} C_VEL
LIN {X 0,Y 493.226,Z 1089.471,A -85,B 0,C 180,E1 6714.457,E2 6714.457} C_VEL
LIN {X 0,Y 490.341,Z 1129.908,A -85,B 0,C 180,E1 6716.123,E2 6716.123} C_VEL
LIN {X 0,Y 486.833,Z 1168.397,A -85,B 0,C 180,E1 6718.472,E2 6718.472} C_VEL
LIN {X 0,Y 483.319,Z 1203.602,A -85,B 0,C 180,E1 6721.428,E2 6721.428} C_VEL
LIN {X 0,Y 479.903,Z 1233.358,A -85,B 0,C 180,E1 6724.881,E2 6724.881} C_VEL
LIN {X 0,Y 477.046,Z 1259.409,A -85,B 0,C 180,E1 6728.86,E2 6728.86} C_VEL
LIN {X 0,Y 475.121,Z 1280.235,A -85,B 0,C 180,E1 6733.084,E2 6733.084} C_VEL
LIN {X 0,Y 474.052,Z 1296.399,A -85,B 0,C 180,E1 6737.592,E2 6737.592} C_VEL
LIN {X 0,Y 473.683,Z 1306.624,A -85,B 0,C 180,E1 6741.772,E2 6741.772} C_VEL
LIN {X 0,Y 473.501,Z 1312.908,A -85,B 0,C 180,E1 6746.345,E2 6746.345} C_VEL
LIN {X 0,Y 473.537,Z 1314.5,A -85,B 0,C 180,E1 6749.999,E2 6749.999} C_VEL
LIN {X 0,Y 473.477,Z 1312.912,A -85,B 0,C 180,E1 6753.654,E2 6753.654} C_VEL
LIN {X 0,Y 473.7,Z 1306.627,A -85,B 0,C 180,E1 6758.228,E2 6758.228} C_VEL
LIN {X 0,Y 474.311,Z 1293.984,A -85,B 0,C 180,E1 6763.192,E2 6763.192} C_VEL
LIN {X 0,Y 475.511,Z 1276.24,A -85,B 0,C 180,E1 6767.826,E2 6767.826} C_VEL
LIN {X 0,Y 477.627,Z 1254.187,A -85,B 0,C 180,E1 6772.029,E2 6772.029} C_VEL
LIN {X 0,Y 480.504,Z 1227.86,A -85,B 0,C 180,E1 6775.832,E2 6775.832} C_VEL
LIN {X 0,Y 483.92,Z 1198.169,A -85,B 0,C 180,E1 6779.096,E2 6779.096} C_VEL
LIN {X 0,Y 487.366,Z 1163.186,A -85,B 0,C 180,E1 6781.89,E2 6781.89} C_VEL
LIN {X 0,Y 490.636,Z 1125.212,A -85,B 0,C 180,E1 6784.11,E2 6784.11} C_VEL
LIN {X 0,Y 493.398,Z 1086.629,A -85,B 0,C 180,E1 6785.624,E2 6785.624} C_VEL
LIN {X 0,Y 495.115,Z 1044.091,A -85,B 0,C 180,E1 6786.562,E2 6786.562} C_VEL
LIN {X 0,Y 494.574,Z 1033.878,A -85,B 0,C 180,E1 6786.785,E2 6786.785} C_VEL
LIN {X 0,Y 472.738,Z 990.374,A -85,B 0,C 180,E1 6789.519,E2 6789.519} C_VEL
LIN {X 0,Y 472.587,Z 989.03,A -85,B 0,C 180,E1 6789.688,E2 6789.688} C_VEL
LIN {X 0,Y 472.478,Z 989.03,A -85,B 0,C 180,E1 6795.363,E2 6795.363} C_VEL
LIN {X 0,Y 472.565,Z 989.03,A -85,B 0,C 180,E1 6800.311,E2 6800.311} C_VEL
LIN {X 0,Y 472.543,Z 989.03,A -85,B 0,C 180,E1 6806.126,E2 6806.126} C_VEL
LIN {X 0,Y 472.659,Z 989.03,A -85,B 0,C 180,E1 6811.388,E2 6811.388} C_VEL
LIN {X 0,Y 472.862,Z 989.03,A -85,B 0,C 180,E1 6817.736,E2 6817.736} C_VEL
LIN {X 0,Y 472.93,Z 989.03,A -85,B 0,C 180,E1 6823.312,E2 6823.312} C_VEL
LIN {X 0,Y 472.981,Z 989.03,A -85,B 0,C 180,E1 6828.964,E2 6828.964} C_VEL
LIN {X 0,Y 473.286,Z 989.03,A -85,B 0,C 180,E1 6834.511,E2 6834.511} C_VEL
LIN {X 0,Y 473.365,Z 989.03,A -85,B 0,C 180,E1 6840,E2 6840} C_VEL
LIN {X 0,Y 473.247,Z 989.03,A -85,B 0,C 180,E1 6845.489,E2 6845.489} C_VEL
LIN {X 0,Y 473.112,Z 989.03,A -85,B 0,C 180,E1 6851.032,E2 6851.032} C_VEL
LIN {X 0,Y 472.954,Z 989.03,A -85,B 0,C 180,E1 6856.829,E2 6856.829} C_VEL
LIN {X 0,Y 472.834,Z 989.03,A -85,B 0,C 180,E1 6862.517,E2 6862.517} C_VEL
LIN {X 0,Y 472.653,Z 989.03,A -85,B 0,C 180,E1 6868.612,E2 6868.612} C_VEL
LIN {X 0,Y 472.547,Z 989.03,A -85,B 0,C 180,E1 6875.084,E2 6875.084} C_VEL
LIN {X 0,Y 472.41,Z 989.03,A -85,B 0,C 180,E1 6882.126,E2 6882.126} C_VEL
LIN {X 0,Y 472.492,Z 989.03,A -85,B 0,C 180,E1 6887.881,E2 6887.881} C_VEL
LIN {X 0,Y 472.67,Z 989.151,A -85,B 0,C 180,E1 6894.568,E2 6894.568} C_VEL
LIN {X 0,Y 482.346,Z 1017.498,A -85,B 0,C 180,E1 6897.635,E2 6897.635} C_VEL
LIN {X 0,Y 485.841,Z 1033.842,A -85,B 0,C 180,E1 6899.446,E2 6899.446} C_VEL
LIN {X 0,Y 481.757,Z 1067.25,A -85,B 0,C 180,E1 6902.852,E2 6902.852} C_VEL
LIN {X 0,Y 478.422,Z 1096.213,A -85,B 0,C 180,E1 6906.659,E2 6906.659} C_VEL
LIN {X 0,Y 476.006,Z 1121.164,A -85,B 0,C 180,E1 6911.039,E2 6911.039} C_VEL
LIN {X 0,Y 474.467,Z 1140.914,A -85,B 0,C 180,E1 6915.828,E2 6915.828} C_VEL
LIN {X 0,Y 473.841,Z 1153.813,A -85,B 0,C 180,E1 6920.376,E2 6920.376} C_VEL
LIN {X 0,Y 473.536,Z 1161.02,A -85,B 0,C 180,E1 6924.515,E2 6924.515} C_VEL
LIN {X 0,Y 473.514,Z 1164.115,A -85,B 0,C 180,E1 6928.174,E2 6928.174} C_VEL
LIN {X 0,Y 473.584,Z 1164.065,A -85,B 0,C 180,E1 6931.827,E2 6931.827} C_VEL
LIN {X 0,Y 473.561,Z 1159.689,A -85,B 0,C 180,E1 6936.404,E2 6936.404} C_VEL
LIN {X 0,Y 473.875,Z 1150.193,A -85,B 0,C 180,E1 6941.016,E2 6941.016} C_VEL
LIN {X 0,Y 474.816,Z 1135.124,A -85,B 0,C 180,E1 6945.673,E2 6945.673} C_VEL
LIN {X 0,Y 476.612,Z 1113.405,A -85,B 0,C 180,E1 6950.382,E2 6950.382} C_VEL
LIN {X 0,Y 479.363,Z 1088.28,A -85,B 0,C 180,E1 6954.405,E2 6954.405} C_VEL
LIN {X 0,Y 482.888,Z 1057.633,A -85,B 0,C 180,E1 6958.129,E2 6958.129} C_VEL
LIN {X 0,Y 485.612,Z 1030.971,A -85,B 0,C 180,E1 6960.772,E2 6960.772} C_VEL
LIN {X 0,Y 477.838,Z 1003.046,A -85,B 0,C 180,E1 6963.853,E2 6963.853} C_VEL
LIN {X 0,Y 472.587,Z 989.03,A -85,B 0,C 180,E1 6965.481,E2 6965.481} C_VEL
LIN {X 0,Y 472.414,Z 989.03,A -85,B 0,C 180,E1 6972.129,E2 6972.129} C_VEL
LIN {X 0,Y 472.492,Z 989.03,A -85,B 0,C 180,E1 6977.883,E2 6977.883} C_VEL
LIN {X 0,Y 472.647,Z 989.03,A -85,B 0,C 180,E1 6982.957,E2 6982.957} C_VEL
LIN {X 0,Y 472.643,Z 989.03,A -85,B 0,C 180,E1 6989.547,E2 6989.547} C_VEL
LIN {X 0,Y 472.78,Z 989.03,A -85,B 0,C 180,E1 6995.486,E2 6995.486} C_VEL
LIN {X 0,Y 472.98,Z 989.03,A -85,B 0,C 180,E1 7001.396,E2 7001.396} C_VEL
LIN {X 0,Y 472.912,Z 989.03,A -85,B 0,C 180,E1 7007.094,E2 7007.094} C_VEL
LIN {X 0,Y 473.219,Z 989.03,A -85,B 0,C 180,E1 7012.979,E2 7012.979} C_VEL
LIN {X 0,Y 473.525,Z 989.03,A -85,B 0,C 180,E1 7018.174,E2 7018.174} C_VEL
LIN {X 0,Y 473.398,Z 989.03,A -85,B 0,C 180,E1 7023.655,E2 7023.655} C_VEL
LIN {X 0,Y 473.207,Z 989.03,A -85,B 0,C 180,E1 7029.174,E2 7029.174} C_VEL
LIN {X 0,Y 473.038,Z 989.03,A -85,B 0,C 180,E1 7034.785,E2 7034.785} C_VEL
LIN {X 0,Y 472.882,Z 989.03,A -85,B 0,C 180,E1 7040.549,E2 7040.549} C_VEL
LIN {X 0,Y 472.707,Z 989.03,A -85,B 0,C 180,E1 7046.639,E2 7046.639} C_VEL
LIN {X 0,Y 472.676,Z 989.03,A -85,B 0,C 180,E1 7052.868,E2 7052.868} C_VEL
LIN {X 0,Y 472.692,Z 989.03,A -85,B 0,C 180,E1 7057.339,E2 7057.339} C_VEL
LIN {X 0,Y 472.445,Z 989.03,A -85,B 0,C 180,E1 7062.723,E2 7062.723} C_VEL
LIN {X 0,Y 472.477,Z 989.03,A -85,B 0,C 180,E1 7067.878,E2 7067.878} C_VEL
LIN {X 0,Y 472.635,Z 989.03,A -85,B 0,C 180,E1 7070.437,E2 7070.437} C_VEL
LIN {X 0,Y 477.102,Z 998.902,A -85,B 0,C 180,E1 7071.053,E2 7071.053} C_VEL
LIN {X 0,Y 495.107,Z 1034.44,A -85,B 0,C 180,E1 7073.269,E2 7073.269} C_VEL
LIN {X 0,Y 494.951,Z 1046.987,A -85,B 0,C 180,E1 7073.475,E2 7073.475} C_VEL
LIN {X 0,Y 491.129,Z 1064.131,A -85,B 0,C 180,E1 7073.521,E2 7073.521} C_VEL
LIN {X 0,Y 487.246,Z 1079.008,A -85,B 0,C 180,E1 7073.641,E2 7073.641} C_VEL
LIN {X 0,Y 487.063,Z 1081.078,A -85,B 0,C 180,E1 7073.698,E2 7073.698} C_VEL
LIN {X 0,Y 484.165,Z 1120.594,A -85,B 0,C 180,E1 7075.197,E2 7075.197} C_VEL
LIN {X 0,Y 480.589,Z 1158.397,A -85,B 0,C 180,E1 7077.356,E2 7077.356} C_VEL
LIN {X 0,Y 476.859,Z 1194.451,A -85,B 0,C 180,E1 7080.208,E2 7080.208} C_VEL
LIN {X 0,Y 473.444,Z 1225.897,A -85,B 0,C 180,E1 7083.498,E2 7083.498} C_VEL
LIN {X 0,Y 470.301,Z 1252.691,A -85,B 0,C 180,E1 7087.353,E2 7087.353} C_VEL
LIN {X 0,Y 467.935,Z 1275.083,A -85,B 0,C 180,E1 7091.616,E2 7091.616} C_VEL
LIN {X 0,Y 466.577,Z 1292.048,A -85,B 0,C 180,E1 7095.983,E2 7095.983} C_VEL
LIN {X 0,Y 465.905,Z 1304.677,A -85,B 0,C 180,E1 7100.68,E2 7100.68} C_VEL
LIN {X 0,Y 465.626,Z 1310.955,A -85,B 0,C 180,E1 7104.42,E2 7104.42} C_VEL
LIN {X 0,Y 465.62,Z 1314.089,A -85,B 0,C 180,E1 7108.142,E2 7108.142} C_VEL
LIN {X 0,Y 465.671,Z 1314.09,A -85,B 0,C 180,E1 7111.856,E2 7111.856} C_VEL
LIN {X 0,Y 465.732,Z 1309.755,A -85,B 0,C 180,E1 7116.511,E2 7116.511} C_VEL
LIN {X 0,Y 466.017,Z 1300.307,A -85,B 0,C 180,E1 7121.202,E2 7121.202} C_VEL
LIN {X 0,Y 467.078,Z 1285.293,A -85,B 0,C 180,E1 7125.938,E2 7125.938} C_VEL
LIN {X 0,Y 469.087,Z 1263.655,A -85,B 0,C 180,E1 7130.723,E2 7130.723} C_VEL
LIN {X 0,Y 471.896,Z 1238.606,A -85,B 0,C 180,E1 7134.815,E2 7134.815} C_VEL
LIN {X 0,Y 474.886,Z 1212.598,A -85,B 0,C 180,E1 7138.013,E2 7138.013} C_VEL
LIN {X 0,Y 478.824,Z 1175.949,A -85,B 0,C 180,E1 7141.369,E2 7141.369} C_VEL
LIN {X 0,Y 482.75,Z 1136.63,A -85,B 0,C 180,E1 7143.981,E2 7143.981} C_VEL
LIN {X 0,Y 486.019,Z 1096.453,A -85,B 0,C 180,E1 7145.807,E2 7145.807} C_VEL
LIN {X 0,Y 488.377,Z 1056.623,A -85,B 0,C 180,E1 7146.875,E2 7146.875} C_VEL
LIN {X 0,Y 488.24,Z 1036.746,A -85,B 0,C 180,E1 7147.267,E2 7147.267} C_VEL
LIN {X 0,Y 466.392,Z 993.957,A -85,B 0,C 180,E1 7150.068,E2 7150.068} C_VEL
LIN {X 0,Y 464.617,Z 989.03,A -85,B 0,C 180,E1 7150.362,E2 7150.362} C_VEL
LIN {X 0,Y 464.591,Z 989.03,A -85,B 0,C 180,E1 7156.995,E2 7156.995} C_VEL
LIN {X 0,Y 464.632,Z 989.03,A -85,B 0,C 180,E1 7161.899,E2 7161.899} C_VEL
LIN {X 0,Y 464.595,Z 989.03,A -85,B 0,C 180,E1 7167.616,E2 7167.616} C_VEL
LIN {X 0,Y 464.769,Z 989.03,A -85,B 0,C 180,E1 7172.965,E2 7172.965} C_VEL
LIN {X 0,Y 464.969,Z 989.03,A -85,B 0,C 180,E1 7179.085,E2 7179.085} C_VEL
LIN {X 0,Y 464.911,Z 989.03,A -85,B 0,C 180,E1 7184.95,E2 7184.95} C_VEL
LIN {X 0,Y 465.144,Z 989.03,A -85,B 0,C 180,E1 7190.665,E2 7190.665} C_VEL
LIN {X 0,Y 465.405,Z 989.03,A -85,B 0,C 180,E1 7196.282,E2 7196.282} C_VEL
LIN {X 0,Y 465.433,Z 989.03,A -85,B 0,C 180,E1 7201.858,E2 7201.858} C_VEL
LIN {X 0,Y 465.282,Z 989.03,A -85,B 0,C 180,E1 7207.454,E2 7207.454} C_VEL
LIN {X 0,Y 465.163,Z 989.03,A -85,B 0,C 180,E1 7213.294,E2 7213.294} C_VEL
LIN {X 0,Y 464.956,Z 989.03,A -85,B 0,C 180,E1 7219.749,E2 7219.749} C_VEL
LIN {X 0,Y 464.844,Z 989.03,A -85,B 0,C 180,E1 7224.961,E2 7224.961} C_VEL
LIN {X 0,Y 464.628,Z 989.03,A -85,B 0,C 180,E1 7231.307,E2 7231.307} C_VEL
LIN {X 0,Y 464.586,Z 989.03,A -85,B 0,C 180,E1 7235.777,E2 7235.777} C_VEL
LIN {X 0,Y 464.483,Z 989.03,A -85,B 0,C 180,E1 7241.65,E2 7241.65} C_VEL
LIN {X 0,Y 464.574,Z 989.03,A -85,B 0,C 180,E1 7248.335,E2 7248.335} C_VEL
LIN {X 0,Y 464.79,Z 989.787,A -85,B 0,C 180,E1 7253.806,E2 7253.806} C_VEL
LIN {X 0,Y 474.925,Z 1017.793,A -85,B 0,C 180,E1 7256.959,E2 7256.959} C_VEL
LIN {X 0,Y 478.89,Z 1037.088,A -85,B 0,C 180,E1 7259.14,E2 7259.14} C_VEL
LIN {X 0,Y 474.933,Z 1066.712,A -85,B 0,C 180,E1 7262.226,E2 7262.226} C_VEL
LIN {X 0,Y 470.588,Z 1099.432,A -85,B 0,C 180,E1 7266.765,E2 7266.765} C_VEL
LIN {X 0,Y 468.115,Z 1123.381,A -85,B 0,C 180,E1 7271.195,E2 7271.195} C_VEL
LIN {X 0,Y 466.558,Z 1142.224,A -85,B 0,C 180,E1 7275.992,E2 7275.992} C_VEL
LIN {X 0,Y 465.902,Z 1154.771,A -85,B 0,C 180,E1 7280.681,E2 7280.681} C_VEL
LIN {X 0,Y 465.648,Z 1161.018,A -85,B 0,C 180,E1 7284.422,E2 7284.422} C_VEL
LIN {X 0,Y 465.615,Z 1164.115,A -85,B 0,C 180,E1 7288.143,E2 7288.143} C_VEL
LIN {X 0,Y 465.693,Z 1164.066,A -85,B 0,C 180,E1 7291.858,E2 7291.858} C_VEL
LIN {X 0,Y 465.661,Z 1159.69,A -85,B 0,C 180,E1 7296.513,E2 7296.513} C_VEL
LIN {X 0,Y 466.014,Z 1150.196,A -85,B 0,C 180,E1 7301.204,E2 7301.204} C_VEL
LIN {X 0,Y 467.063,Z 1135.128,A -85,B 0,C 180,E1 7305.94,E2 7305.94} C_VEL
LIN {X 0,Y 469.008,Z 1113.408,A -85,B 0,C 180,E1 7310.728,E2 7310.728} C_VEL
LIN {X 0,Y 471.948,Z 1088.285,A -85,B 0,C 180,E1 7314.814,E2 7314.814} C_VEL
LIN {X 0,Y 475.984,Z 1059.314,A -85,B 0,C 180,E1 7318.538,E2 7318.538} C_VEL
LIN {X 0,Y 478.974,Z 1034.723,A -85,B 0,C 180,E1 7321.003,E2 7321.003} C_VEL
LIN {X 0,Y 471.507,Z 1007.075,A -85,B 0,C 180,E1 7324.163,E2 7324.163} C_VEL
LIN {X 0,Y 464.643,Z 989.03,A -85,B 0,C 180,E1 7326.267,E2 7326.267} C_VEL
LIN {X 0,Y 464.534,Z 989.03,A -85,B 0,C 180,E1 7333.015,E2 7333.015} C_VEL
LIN {X 0,Y 464.582,Z 989.03,A -85,B 0,C 180,E1 7339.489,E2 7339.489} C_VEL
LIN {X 0,Y 464.688,Z 989.03,A -85,B 0,C 180,E1 7344.277,E2 7344.277} C_VEL
LIN {X 0,Y 464.758,Z 989.03,A -85,B 0,C 180,E1 7351.243,E2 7351.243} C_VEL
LIN {X 0,Y 464.878,Z 989.03,A -85,B 0,C 180,E1 7357.076,E2 7357.076} C_VEL
LIN {X 0,Y 465.048,Z 989.03,A -85,B 0,C 180,E1 7363.021,E2 7363.021} C_VEL
LIN {X 0,Y 465.059,Z 989.03,A -85,B 0,C 180,E1 7368.774,E2 7368.774} C_VEL
LIN {X 0,Y 465.406,Z 989.03,A -85,B 0,C 180,E1 7374.418,E2 7374.418} C_VEL
LIN {X 0,Y 465.576,Z 989.03,A -85,B 0,C 180,E1 7380,E2 7380} C_VEL
LIN {X 0,Y 465.372,Z 989.03,A -85,B 0,C 180,E1 7385.582,E2 7385.582} C_VEL
LIN {X 0,Y 465.197,Z 989.03,A -85,B 0,C 180,E1 7391.223,E2 7391.223} C_VEL
LIN {X 0,Y 465.046,Z 989.03,A -85,B 0,C 180,E1 7396.979,E2 7396.979} C_VEL
LIN {X 0,Y 464.867,Z 989.03,A -85,B 0,C 180,E1 7402.924,E2 7402.924} C_VEL
LIN {X 0,Y 464.756,Z 989.03,A -85,B 0,C 180,E1 7409.144,E2 7409.144} C_VEL
LIN {X 0,Y 464.772,Z 989.03,A -85,B 0,C 180,E1 7415.76,E2 7415.76} C_VEL
LIN {X 0,Y 464.536,Z 989.03,A -85,B 0,C 180,E1 7421.656,E2 7421.656} C_VEL
LIN {X 0,Y 464.575,Z 989.03,A -85,B 0,C 180,E1 7428.335,E2 7428.335} C_VEL
LIN {X 0,Y 464.635,Z 989.03,A -85,B 0,C 180,E1 7429.639,E2 7429.639} C_VEL
LIN {X 0,Y 469.38,Z 999.199,A -85,B 0,C 180,E1 7430.326,E2 7430.326} C_VEL
LIN {X 0,Y 488.653,Z 1037.159,A -85,B 0,C 180,E1 7432.776,E2 7432.776} C_VEL
LIN {X 0,Y 487.063,Z 1081.078,A -85,B 0,C 180,E1 7433.698,E2 7433.698} C_VEL
LIN {X 0,Y 482.627,Z 1097.914,A -85,B 0,C 180,E1 7433.984,E2 7433.984} C_VEL
LIN {X 0,Y 478.161,Z 1112.332,A -85,B 0,C 180,E1 7434.317,E2 7434.317} C_VEL
LIN {X 0,Y 477.909,Z 1114.369,A -85,B 0,C 180,E1 7434.407,E2 7434.407} C_VEL
LIN {X 0,Y 473.958,Z 1154.43,A -85,B 0,C 180,E1 7436.646,E2 7436.646} C_VEL
LIN {X 0,Y 469.944,Z 1190.32,A -85,B 0,C 180,E1 7439.457,E2 7439.457} C_VEL
LIN {X 0,Y 466.223,Z 1222.796,A -85,B 0,C 180,E1 7442.828,E2 7442.828} C_VEL
LIN {X 0,Y 463.222,Z 1248.812,A -85,B 0,C 180,E1 7446.313,E2 7446.313} C_VEL
LIN {X 0,Y 460.475,Z 1273.174,A -85,B 0,C 180,E1 7450.87,E2 7450.87} C_VEL
LIN {X 0,Y 458.763,Z 1292.047,A -85,B 0,C 180,E1 7455.739,E2 7455.739} C_VEL
LIN {X 0,Y 458.029,Z 1304.677,A -85,B 0,C 180,E1 7460.518,E2 7460.518} C_VEL
LIN {X 0,Y 457.733,Z 1310.954,A -85,B 0,C 180,E1 7464.323,E2 7464.323} C_VEL
LIN {X 0,Y 457.715,Z 1314.089,A -85,B 0,C 180,E1 7468.11,E2 7468.11} C_VEL
LIN {X 0,Y 457.765,Z 1314.09,A -85,B 0,C 180,E1 7471.888,E2 7471.888} C_VEL
LIN {X 0,Y 457.841,Z 1309.755,A -85,B 0,C 180,E1 7476.624,E2 7476.624} C_VEL
LIN {X 0,Y 458.188,Z 1300.308,A -85,B 0,C 180,E1 7481.396,E2 7481.396} C_VEL
LIN {X 0,Y 459.325,Z 1285.294,A -85,B 0,C 180,E1 7486.215,E2 7486.215} C_VEL
LIN {X 0,Y 461.481,Z 1263.653,A -85,B 0,C 180,E1 7491.081,E2 7491.081} C_VEL
LIN {X 0,Y 464.239,Z 1239.928,A -85,B 0,C 180,E1 7494.996,E2 7494.996} C_VEL
LIN {X 0,Y 468.023,Z 1207.043,A -85,B 0,C 180,E1 7498.922,E2 7498.922} C_VEL
LIN {X 0,Y 472.124,Z 1171.635,A -85,B 0,C 180,E1 7502.107,E2 7502.107} C_VEL
LIN {X 0,Y 476.1,Z 1133.478,A -85,B 0,C 180,E1 7504.628,E2 7504.628} C_VEL
LIN {X 0,Y 479.494,Z 1095.028,A -85,B 0,C 180,E1 7506.372,E2 7506.372} C_VEL
LIN {X 0,Y 482.002,Z 1055.088,A -85,B 0,C 180,E1 7507.448,E2 7507.448} C_VEL
LIN {X 0,Y 481.612,Z 1038.952,A -85,B 0,C 180,E1 7507.802,E2 7507.802} C_VEL
LIN {X 0,Y 461.043,Z 998.697,A -85,B 0,C 180,E1 7510.512,E2 7510.512} C_VEL
LIN {X 0,Y 456.677,Z 989.03,A -85,B 0,C 180,E1 7511.212,E2 7511.212} C_VEL
LIN {X 0,Y 456.683,Z 989.03,A -85,B 0,C 180,E1 7516.63,E2 7516.63} C_VEL
LIN {X 0,Y 456.692,Z 989.03,A -85,B 0,C 180,E1 7522.467,E2 7522.467} C_VEL
LIN {X 0,Y 456.687,Z 989.03,A -85,B 0,C 180,E1 7529.215,E2 7529.215} C_VEL
LIN {X 0,Y 456.851,Z 989.03,A -85,B 0,C 180,E1 7534.572,E2 7534.572} C_VEL
LIN {X 0,Y 457.083,Z 989.03,A -85,B 0,C 180,E1 7540.724,E2 7540.724} C_VEL
LIN {X 0,Y 457.082,Z 989.03,A -85,B 0,C 180,E1 7546.639,E2 7546.639} C_VEL
LIN {X 0,Y 457.384,Z 989.03,A -85,B 0,C 180,E1 7552.417,E2 7552.417} C_VEL
LIN {X 0,Y 457.699,Z 989.03,A -85,B 0,C 180,E1 7558.111,E2 7558.111} C_VEL
LIN {X 0,Y 457.572,Z 989.03,A -85,B 0,C 180,E1 7563.782,E2 7563.782} C_VEL
LIN {X 0,Y 457.374,Z 989.03,A -85,B 0,C 180,E1 7569.495,E2 7569.495} C_VEL
LIN {X 0,Y 457.158,Z 989.03,A -85,B 0,C 180,E1 7575.311,E2 7575.311} C_VEL
LIN {X 0,Y 457.004,Z 989.03,A -85,B 0,C 180,E1 7581.297,E2 7581.297} C_VEL
LIN {X 0,Y 456.823,Z 989.03,A -85,B 0,C 180,E1 7587.544,E2 7587.544} C_VEL
LIN {X 0,Y 456.628,Z 989.03,A -85,B 0,C 180,E1 7594.294,E2 7594.294} C_VEL
LIN {X 0,Y 456.573,Z 989.03,A -85,B 0,C 180,E1 7600.522,E2 7600.522} C_VEL
LIN {X 0,Y 456.679,Z 989.03,A -85,B 0,C 180,E1 7606.628,E2 7606.628} C_VEL
LIN {X 0,Y 456.838,Z 989.545,A -85,B 0,C 180,E1 7612.946,E2 7612.946} C_VEL
LIN {X 0,Y 468.093,Z 1020.085,A -85,B 0,C 180,E1 7616.489,E2 7616.489} C_VEL
LIN {X 0,Y 471.955,Z 1040.424,A -85,B 0,C 180,E1 7618.835,E2 7618.835} C_VEL
LIN {X 0,Y 467.674,Z 1070.72,A -85,B 0,C 180,E1 7622.105,E2 7622.105} C_VEL
LIN {X 0,Y 463.455,Z 1098.127,A -85,B 0,C 180,E1 7626.073,E2 7626.073} C_VEL
LIN {X 0,Y 460.445,Z 1123.377,A -85,B 0,C 180,E1 7630.87,E2 7630.87} C_VEL
LIN {X 0,Y 458.743,Z 1142.221,A -85,B 0,C 180,E1 7635.748,E2 7635.748} C_VEL
LIN {X 0,Y 458.026,Z 1154.77,A -85,B 0,C 180,E1 7640.519,E2 7640.519} C_VEL
LIN {X 0,Y 457.754,Z 1161.017,A -85,B 0,C 180,E1 7644.325,E2 7644.325} C_VEL
LIN {X 0,Y 457.71,Z 1164.115,A -85,B 0,C 180,E1 7648.111,E2 7648.111} C_VEL
LIN {X 0,Y 457.787,Z 1164.066,A -85,B 0,C 180,E1 7651.89,E2 7651.89} C_VEL
LIN {X 0,Y 457.775,Z 1159.691,A -85,B 0,C 180,E1 7656.626,E2 7656.626} C_VEL
LIN {X 0,Y 458.182,Z 1150.198,A -85,B 0,C 180,E1 7661.398,E2 7661.398} C_VEL
LIN {X 0,Y 459.31,Z 1135.132,A -85,B 0,C 180,E1 7666.217,E2 7666.217} C_VEL
LIN {X 0,Y 461.45,Z 1113.411,A -85,B 0,C 180,E1 7671.084,E2 7671.084} C_VEL
LIN {X 0,Y 465.31,Z 1086.182,A -85,B 0,C 180,E1 7675.707,E2 7675.707} C_VEL
LIN {X 0,Y 469.484,Z 1058.074,A -85,B 0,C 180,E1 7679.29,E2 7679.29} C_VEL
LIN {X 0,Y 472.187,Z 1037.928,A -85,B 0,C 180,E1 7681.312,E2 7681.312} C_VEL
LIN {X 0,Y 465.334,Z 1011.423,A -85,B 0,C 180,E1 7684.441,E2 7684.441} C_VEL
LIN {X 0,Y 456.694,Z 989.03,A -85,B 0,C 180,E1 7687.052,E2 7687.052} C_VEL
LIN {X 0,Y 456.599,Z 989.03,A -85,B 0,C 180,E1 7693.951,E2 7693.951} C_VEL
LIN {X 0,Y 456.692,Z 989.03,A -85,B 0,C 180,E1 7699.463,E2 7699.463} C_VEL
LIN {X 0,Y 456.676,Z 989.03,A -85,B 0,C 180,E1 7705.826,E2 7705.826} C_VEL
LIN {X 0,Y 456.833,Z 989.03,A -85,B 0,C 180,E1 7712.456,E2 7712.456} C_VEL
LIN {X 0,Y 457.02,Z 989.03,A -85,B 0,C 180,E1 7718.704,E2 7718.704} C_VEL
LIN {X 0,Y 457.013,Z 989.03,A -85,B 0,C 180,E1 7724.684,E2 7724.684} C_VEL
LIN {X 0,Y 457.281,Z 989.03,A -85,B 0,C 180,E1 7730.503,E2 7730.503} C_VEL
LIN {X 0,Y 457.507,Z 989.03,A -85,B 0,C 180,E1 7736.218,E2 7736.218} C_VEL
LIN {X 0,Y 457.518,Z 989.03,A -85,B 0,C 180,E1 7741.89,E2 7741.89} C_VEL
LIN {X 0,Y 457.346,Z 989.03,A -85,B 0,C 180,E1 7748.166,E2 7748.166} C_VEL
LIN {X 0,Y 457.282,Z 989.03,A -85,B 0,C 180,E1 7753.355,E2 7753.355} C_VEL
LIN {X 0,Y 457.055,Z 989.03,A -85,B 0,C 180,E1 7759.278,E2 7759.278} C_VEL
LIN {X 0,Y 456.854,Z 989.03,A -85,B 0,C 180,E1 7765.428,E2 7765.428} C_VEL
LIN {X 0,Y 456.801,Z 989.03,A -85,B 0,C 180,E1 7771.906,E2 7771.906} C_VEL
LIN {X 0,Y 456.728,Z 989.03,A -85,B 0,C 180,E1 7778.883,E2 7778.883} C_VEL
LIN {X 0,Y 456.633,Z 989.03,A -85,B 0,C 180,E1 7786.053,E2 7786.053} C_VEL
LIN {X 0,Y 456.666,Z 989.03,A -85,B 0,C 180,E1 7788.846,E2 7788.846} C_VEL
LIN {X 0,Y 460.785,Z 998.22,A -85,B 0,C 180,E1 7789.454,E2 7789.454} C_VEL
LIN {X 0,Y 482.237,Z 1039.643,A -85,B 0,C 180,E1 7792.265,E2 7792.265} C_VEL
LIN {X 0,Y 480.377,Z 1083.373,A -85,B 0,C 180,E1 7793.24,E2 7793.24} C_VEL
LIN {X 0,Y 477.909,Z 1114.369,A -85,B 0,C 180,E1 7794.407,E2 7794.407} C_VEL
LIN {X 0,Y 473.075,Z 1130.792,A -85,B 0,C 180,E1 7794.992,E2 7794.992} C_VEL
LIN {X 0,Y 467.894,Z 1146.349,A -85,B 0,C 180,E1 7795.659,E2 7795.659} C_VEL
LIN {X 0,Y 463.501,Z 1183.629,A -85,B 0,C 180,E1 7798.464,E2 7798.464} C_VEL
LIN {X 0,Y 459.105,Z 1219.023,A -85,B 0,C 180,E1 7802.07,E2 7802.07} C_VEL
LIN {X 0,Y 455.378,Z 1249.948,A -85,B 0,C 180,E1 7806.269,E2 7806.269} C_VEL
LIN {X 0,Y 453.018,Z 1270.987,A -85,B 0,C 180,E1 7810.049,E2 7810.049} C_VEL
LIN {X 0,Y 451.113,Z 1290.312,A -85,B 0,C 180,E1 7814.931,E2 7814.931} C_VEL
LIN {X 0,Y 450.23,Z 1303.716,A -85,B 0,C 180,E1 7819.865,E2 7819.865} C_VEL
LIN {X 0,Y 449.856,Z 1310.954,A -85,B 0,C 180,E1 7824.224,E2 7824.224} C_VEL
LIN {X 0,Y 449.834,Z 1314.089,A -85,B 0,C 180,E1 7828.077,E2 7828.077} C_VEL
LIN {X 0,Y 449.877,Z 1314.091,A -85,B 0,C 180,E1 7831.922,E2 7831.922} C_VEL
LIN {X 0,Y 449.937,Z 1309.754,A -85,B 0,C 180,E1 7836.74,E2 7836.74} C_VEL
LIN {X 0,Y 450.335,Z 1300.308,A -85,B 0,C 180,E1 7841.598,E2 7841.598} C_VEL
LIN {X 0,Y 451.563,Z 1285.293,A -85,B 0,C 180,E1 7846.501,E2 7846.501} C_VEL
LIN {X 0,Y 453.771,Z 1264.588,A -85,B 0,C 180,E1 7851.256,E2 7851.256} C_VEL
LIN {X 0,Y 456.946,Z 1236.742,A -85,B 0,C 180,E1 7855.668,E2 7855.668} C_VEL
LIN {X 0,Y 460.961,Z 1204.05,A -85,B 0,C 180,E1 7859.578,E2 7859.578} C_VEL
LIN {X 0,Y 465.207,Z 1169.803,A -85,B 0,C 180,E1 7862.676,E2 7862.676} C_VEL
LIN {X 0,Y 469.361,Z 1132.286,A -85,B 0,C 180,E1 7865.182,E2 7865.182} C_VEL
LIN {X 0,Y 473.062,Z 1093.492,A -85,B 0,C 180,E1 7866.953,E2 7866.953} C_VEL
LIN {X 0,Y 475.68,Z 1053.676,A -85,B 0,C 180,E1 7868.034,E2 7868.034} C_VEL
LIN {X 0,Y 475.349,Z 1041.909,A -85,B 0,C 180,E1 7868.309,E2 7868.309} C_VEL
LIN {X 0,Y 453.918,Z 999.801,A -85,B 0,C 180,E1 7871.229,E2 7871.229} C_VEL
LIN {X 0,Y 448.809,Z 990.14,A -85,B 0,C 180,E1 7871.978,E2 7871.978} C_VEL
LIN {X 0,Y 448.713,Z 989.03,A -85,B 0,C 180,E1 7872.029,E2 7872.029} C_VEL
LIN {X 0,Y 448.722,Z 989.03,A -85,B 0,C 180,E1 7877.736,E2 7877.736} C_VEL
LIN {X 0,Y 448.745,Z 989.03,A -85,B 0,C 180,E1 7883.808,E2 7883.808} C_VEL
LIN {X 0,Y 448.788,Z 989.03,A -85,B 0,C 180,E1 7889.712,E2 7889.712} C_VEL
LIN {X 0,Y 448.963,Z 989.03,A -85,B 0,C 180,E1 7896.214,E2 7896.214} C_VEL
LIN {X 0,Y 449.15,Z 989.03,A -85,B 0,C 180,E1 7902.401,E2 7902.401} C_VEL
LIN {X 0,Y 449.204,Z 989.03,A -85,B 0,C 180,E1 7908.372,E2 7908.372} C_VEL
LIN {X 0,Y 449.586,Z 989.03,A -85,B 0,C 180,E1 7914.221,E2 7914.221} C_VEL
LIN {X 0,Y 449.707,Z 989.03,A -85,B 0,C 180,E1 7920,E2 7920} C_VEL
LIN {X 0,Y 449.533,Z 989.03,A -85,B 0,C 180,E1 7925.779,E2 7925.779} C_VEL
LIN {X 0,Y 449.348,Z 989.03,A -85,B 0,C 180,E1 7931.624,E2 7931.624} C_VEL
LIN {X 0,Y 449.165,Z 989.03,A -85,B 0,C 180,E1 7937.599,E2 7937.599} C_VEL
LIN {X 0,Y 448.974,Z 989.03,A -85,B 0,C 180,E1 7943.785,E2 7943.785} C_VEL
LIN {X 0,Y 448.79,Z 989.03,A -85,B 0,C 180,E1 7950.287,E2 7950.287} C_VEL
LIN {X 0,Y 448.653,Z 989.03,A -85,B 0,C 180,E1 7957.257,E2 7957.257} C_VEL
LIN {X 0,Y 448.648,Z 989.03,A -85,B 0,C 180,E1 7962.273,E2 7962.273} C_VEL
LIN {X 0,Y 448.72,Z 989.03,A -85,B 0,C 180,E1 7967.734,E2 7967.734} C_VEL
LIN {X 0,Y 448.854,Z 989.387,A -85,B 0,C 180,E1 7972.045,E2 7972.045} C_VEL
LIN {X 0,Y 460.76,Z 1020.697,A -85,B 0,C 180,E1 7975.8,E2 7975.8} C_VEL
LIN {X 0,Y 465.147,Z 1042.942,A -85,B 0,C 180,E1 7978.445,E2 7978.445} C_VEL
LIN {X 0,Y 460.368,Z 1074.662,A -85,B 0,C 180,E1 7981.969,E2 7981.969} C_VEL
LIN {X 0,Y 455.989,Z 1101.458,A -85,B 0,C 180,E1 7986.013,E2 7986.013} C_VEL
LIN {X 0,Y 452.774,Z 1123.418,A -85,B 0,C 180,E1 7990.533,E2 7990.533} C_VEL
LIN {X 0,Y 450.958,Z 1141.866,A -85,B 0,C 180,E1 7995.383,E2 7995.383} C_VEL
LIN {X 0,Y 450.151,Z 1154.768,A -85,B 0,C 180,E1 8000.352,E2 8000.352} C_VEL
LIN {X 0,Y 449.874,Z 1161.016,A -85,B 0,C 180,E1 8004.225,E2 8004.225} C_VEL
LIN {X 0,Y 449.829,Z 1164.115,A -85,B 0,C 180,E1 8008.078,E2 8008.078} C_VEL
LIN {X 0,Y 449.897,Z 1164.067,A -85,B 0,C 180,E1 8011.923,E2 8011.923} C_VEL
LIN {X 0,Y 449.873,Z 1159.692,A -85,B 0,C 180,E1 8016.743,E2 8016.743} C_VEL
LIN {X 0,Y 450.329,Z 1150.2,A -85,B 0,C 180,E1 8021.599,E2 8021.599} C_VEL
LIN {X 0,Y 451.552,Z 1135.135,A -85,B 0,C 180,E1 8026.503,E2 8026.503} C_VEL
LIN {X 0,Y 454.784,Z 1109.35,A -85,B 0,C 180,E1 8032.431,E2 8032.431} C_VEL
LIN {X 0,Y 458.795,Z 1084.299,A -85,B 0,C 180,E1 8036.625,E2 8036.625} C_VEL
LIN {X 0,Y 463.59,Z 1054.036,A -85,B 0,C 180,E1 8040.349,E2 8040.349} C_VEL
LIN {X 0,Y 464.976,Z 1038.742,A -85,B 0,C 180,E1 8041.928,E2 8041.928} C_VEL
LIN {X 0,Y 458.324,Z 1013.566,A -85,B 0,C 180,E1 8044.994,E2 8044.994} C_VEL
LIN {X 0,Y 448.717,Z 989.03,A -85,B 0,C 180,E1 8047.907,E2 8047.907} C_VEL
LIN {X 0,Y 448.649,Z 989.03,A -85,B 0,C 180,E1 8054.938,E2 8054.938} C_VEL
LIN {X 0,Y 448.778,Z 989.03,A -85,B 0,C 180,E1 8060.659,E2 8060.659} C_VEL
LIN {X 0,Y 448.717,Z 989.03,A -85,B 0,C 180,E1 8067.449,E2 8067.449} C_VEL
LIN {X 0,Y 448.939,Z 989.03,A -85,B 0,C 180,E1 8074.091,E2 8074.091} C_VEL
LIN {X 0,Y 449.145,Z 989.03,A -85,B 0,C 180,E1 8080.369,E2 8080.369} C_VEL
LIN {X 0,Y 449.181,Z 989.03,A -85,B 0,C 180,E1 8086.972,E2 8086.972} C_VEL
LIN {X 0,Y 449.477,Z 989.03,A -85,B 0,C 180,E1 8092.975,E2 8092.975} C_VEL
LIN {X 0,Y 449.827,Z 989.03,A -85,B 0,C 180,E1 8098.078,E2 8098.078} C_VEL
LIN {X 0,Y 449.67,Z 989.03,A -85,B 0,C 180,E1 8103.848,E2 8103.848} C_VEL
LIN {X 0,Y 449.453,Z 989.03,A -85,B 0,C 180,E1 8109.664,E2 8109.664} C_VEL
LIN {X 0,Y 449.263,Z 989.03,A -85,B 0,C 180,E1 8115.587,E2 8115.587} C_VEL
LIN {X 0,Y 449.069,Z 989.03,A -85,B 0,C 180,E1 8121.692,E2 8121.692} C_VEL
LIN {X 0,Y 448.869,Z 989.03,A -85,B 0,C 180,E1 8128.075,E2 8128.075} C_VEL
LIN {X 0,Y 448.824,Z 989.03,A -85,B 0,C 180,E1 8134.858,E2 8134.858} C_VEL
LIN {X 0,Y 448.757,Z 989.03,A -85,B 0,C 180,E1 8139.708,E2 8139.708} C_VEL
LIN {X 0,Y 448.636,Z 989.03,A -85,B 0,C 180,E1 8145.061,E2 8145.061} C_VEL
LIN {X 0,Y 448.721,Z 989.03,A -85,B 0,C 180,E1 8147.97,E2 8147.97} C_VEL
LIN {X 0,Y 453.214,Z 998.853,A -85,B 0,C 180,E1 8148.68,E2 8148.68} C_VEL
LIN {X 0,Y 474.379,Z 1039.301,A -85,B 0,C 180,E1 8151.554,E2 8151.554} C_VEL
LIN {X 0,Y 475.874,Z 1042.385,A -85,B 0,C 180,E1 8151.747,E2 8151.747} C_VEL
LIN {X 0,Y 473.664,Z 1086.222,A -85,B 0,C 180,E1 8152.79,E2 8152.79} C_VEL
LIN {X 0,Y 470.129,Z 1126.3,A -85,B 0,C 180,E1 8154.498,E2 8154.498} C_VEL
LIN {X 0,Y 467.894,Z 1146.349,A -85,B 0,C 180,E1 8155.659,E2 8155.659} C_VEL
LIN {X 0,Y 462.602,Z 1161.729,A -85,B 0,C 180,E1 8156.475,E2 8156.475} C_VEL
LIN {X 0,Y 457.211,Z 1176.493,A -85,B 0,C 180,E1 8157.433,E2 8157.433} C_VEL
LIN {X 0,Y 452.597,Z 1210.943,A -85,B 0,C 180,E1 8160.815,E2 8160.815} C_VEL
LIN {X 0,Y 448.63,Z 1241.743,A -85,B 0,C 180,E1 8164.811,E2 8164.811} C_VEL
LIN {X 0,Y 445.527,Z 1267.966,A -85,B 0,C 180,E1 8169.277,E2 8169.277} C_VEL
LIN {X 0,Y 443.721,Z 1285.284,A -85,B 0,C 180,E1 8173.197,E2 8173.197} C_VEL
LIN {X 0,Y 442.504,Z 1300.305,A -85,B 0,C 180,E1 8178.193,E2 8178.193} C_VEL
LIN {X 0,Y 442.071,Z 1309.748,A -85,B 0,C 180,E1 8183.138,E2 8183.138} C_VEL
LIN {X 0,Y 441.929,Z 1314.089,A -85,B 0,C 180,E1 8188.042,E2 8188.042} C_VEL
LIN {X 0,Y 441.971,Z 1314.091,A -85,B 0,C 180,E1 8191.956,E2 8191.956} C_VEL
LIN {X 0,Y 442.068,Z 1309.754,A -85,B 0,C 180,E1 8196.861,E2 8196.861} C_VEL
LIN {X 0,Y 442.485,Z 1300.308,A -85,B 0,C 180,E1 8201.806,E2 8201.806} C_VEL
LIN {X 0,Y 443.833,Z 1285.292,A -85,B 0,C 180,E1 8206.797,E2 8206.797} C_VEL
LIN {X 0,Y 445.693,Z 1266.505,A -85,B 0,C 180,E1 8211.007,E2 8211.007} C_VEL
LIN {X 0,Y 448.753,Z 1240.587,A -85,B 0,C 180,E1 8215.361,E2 8215.361} C_VEL
LIN {X 0,Y 452.721,Z 1209.838,A -85,B 0,C 180,E1 8219.311,E2 8219.311} C_VEL
LIN {X 0,Y 457.379,Z 1174.908,A -85,B 0,C 180,E1 8222.705,E2 8222.705} C_VEL
LIN {X 0,Y 462.159,Z 1136.183,A -85,B 0,C 180,E1 8225.462,E2 8225.462} C_VEL
LIN {X 0,Y 466.407,Z 1094.754,A -85,B 0,C 180,E1 8227.452,E2 8227.452} C_VEL
LIN {X 0,Y 469.374,Z 1052.869,A -85,B 0,C 180,E1 8228.625,E2 8228.625} C_VEL
LIN {X 0,Y 468.803,Z 1044.109,A -85,B 0,C 180,E1 8228.874,E2 8228.874} C_VEL
LIN {X 0,Y 448.837,Z 1004.863,A -85,B 0,C 180,E1 8231.671,E2 8231.671} C_VEL
LIN {X 0,Y 440.759,Z 989.597,A -85,B 0,C 180,E1 8232.898,E2 8232.898} C_VEL
LIN {X 0,Y 440.747,Z 989.03,A -85,B 0,C 180,E1 8239.422,E2 8239.422} C_VEL
LIN {X 0,Y 440.812,Z 989.03,A -85,B 0,C 180,E1 8245.242,E2 8245.242} C_VEL
LIN {X 0,Y 440.926,Z 989.03,A -85,B 0,C 180,E1 8251.373,E2 8251.373} C_VEL
LIN {X 0,Y 441.103,Z 989.03,A -85,B 0,C 180,E1 8257.896,E2 8257.896} C_VEL
LIN {X 0,Y 441.174,Z 989.03,A -85,B 0,C 180,E1 8264.12,E2 8264.12} C_VEL
LIN {X 0,Y 441.388,Z 989.03,A -85,B 0,C 180,E1 8270.158,E2 8270.158} C_VEL
LIN {X 0,Y 441.678,Z 989.03,A -85,B 0,C 180,E1 8276.082,E2 8276.082} C_VEL
LIN {X 0,Y 441.739,Z 989.03,A -85,B 0,C 180,E1 8281.958,E2 8281.958} C_VEL
LIN {X 0,Y 441.548,Z 989.03,A -85,B 0,C 180,E1 8287.857,E2 8287.857} C_VEL
LIN {X 0,Y 441.408,Z 989.03,A -85,B 0,C 180,E1 8293.845,E2 8293.845} C_VEL
LIN {X 0,Y 441.186,Z 989.03,A -85,B 0,C 180,E1 8300,E2 8300} C_VEL
LIN {X 0,Y 440.964,Z 989.03,A -85,B 0,C 180,E1 8306.414,E2 8306.414} C_VEL
LIN {X 0,Y 440.743,Z 989.03,A -85,B 0,C 180,E1 8313.215,E2 8313.215} C_VEL
LIN {X 0,Y 440.713,Z 989.03,A -85,B 0,C 180,E1 8318.046,E2 8318.046} C_VEL
LIN {X 0,Y 440.652,Z 989.03,A -85,B 0,C 180,E1 8324.017,E2 8324.017} C_VEL
LIN {X 0,Y 440.912,Z 989.591,A -85,B 0,C 180,E1 8331.128,E2 8331.128} C_VEL
LIN {X 0,Y 452.941,Z 1020.251,A -85,B 0,C 180,E1 8334.931,E2 8334.931} C_VEL
LIN {X 0,Y 458.507,Z 1044.308,A -85,B 0,C 180,E1 8337.934,E2 8337.934} C_VEL
LIN {X 0,Y 453.436,Z 1076.338,A -85,B 0,C 180,E1 8341.545,E2 8341.545} C_VEL
LIN {X 0,Y 448.688,Z 1103.654,A -85,B 0,C 180,E1 8345.757,E2 8345.757} C_VEL
LIN {X 0,Y 445.362,Z 1124.804,A -85,B 0,C 180,E1 8350.195,E2 8350.195} C_VEL
LIN {X 0,Y 442.972,Z 1144.112,A -85,B 0,C 180,E1 8355.853,E2 8355.853} C_VEL
LIN {X 0,Y 442.18,Z 1156.6,A -85,B 0,C 180,E1 8361.123,E2 8361.123} C_VEL
LIN {X 0,Y 441.887,Z 1162.951,A -85,B 0,C 180,E1 8366.084,E2 8366.084} C_VEL
LIN {X 0,Y 441.945,Z 1164.497,A -85,B 0,C 180,E1 8370.001,E2 8370.001} C_VEL
LIN {X 0,Y 441.9,Z 1162.871,A -85,B 0,C 180,E1 8373.917,E2 8373.917} C_VEL
LIN {X 0,Y 442.166,Z 1156.482,A -85,B 0,C 180,E1 8378.85,E2 8378.85} C_VEL
LIN {X 0,Y 442.912,Z 1144.9,A -85,B 0,C 180,E1 8383.798,E2 8383.798} C_VEL
LIN {X 0,Y 445.056,Z 1126.401,A -85,B 0,C 180,E1 8389.318,E2 8389.318} C_VEL
LIN {X 0,Y 448.42,Z 1105.442,A -85,B 0,C 180,E1 8393.818,E2 8393.818} C_VEL
LIN {X 0,Y 452.722,Z 1080.315,A -85,B 0,C 180,E1 8397.818,E2 8397.818} C_VEL
LIN {X 0,Y 457.576,Z 1050.924,A -85,B 0,C 180,E1 8401.308,E2 8401.308} C_VEL
LIN {X 0,Y 458.103,Z 1041.276,A -85,B 0,C 180,E1 8402.346,E2 8402.346} C_VEL
LIN {X 0,Y 452.202,Z 1018.042,A -85,B 0,C 180,E1 8405.263,E2 8405.263} C_VEL
LIN {X 0,Y 440.776,Z 989.03,A -85,B 0,C 180,E1 8408.942,E2 8408.942} C_VEL
LIN {X 0,Y 440.674,Z 989.03,A -85,B 0,C 180,E1 8415.982,E2 8415.982} C_VEL
LIN {X 0,Y 440.822,Z 989.03,A -85,B 0,C 180,E1 8421.965,E2 8421.965} C_VEL
LIN {X 0,Y 440.771,Z 989.03,A -85,B 0,C 180,E1 8426.787,E2 8426.787} C_VEL
LIN {X 0,Y 440.961,Z 989.03,A -85,B 0,C 180,E1 8433.586,E2 8433.586} C_VEL
LIN {X 0,Y 441.213,Z 989.03,A -85,B 0,C 180,E1 8440.001,E2 8440.001} C_VEL
LIN {X 0,Y 441.223,Z 989.03,A -85,B 0,C 180,E1 8446.149,E2 8446.149} C_VEL
LIN {X 0,Y 441.584,Z 989.03,A -85,B 0,C 180,E1 8452.976,E2 8452.976} C_VEL
LIN {X 0,Y 441.879,Z 989.03,A -85,B 0,C 180,E1 8460,E2 8460} C_VEL
LIN {X 0,Y 441.649,Z 989.03,A -85,B 0,C 180,E1 8465.883,E2 8465.883} C_VEL
LIN {X 0,Y 441.452,Z 989.03,A -85,B 0,C 180,E1 8471.835,E2 8471.835} C_VEL
LIN {X 0,Y 441.233,Z 989.03,A -85,B 0,C 180,E1 8477.926,E2 8477.926} C_VEL
LIN {X 0,Y 441.04,Z 989.03,A -85,B 0,C 180,E1 8484.24,E2 8484.24} C_VEL
LIN {X 0,Y 440.88,Z 989.03,A -85,B 0,C 180,E1 8491.163,E2 8491.163} C_VEL
LIN {X 0,Y 440.899,Z 989.03,A -85,B 0,C 180,E1 8495.578,E2 8495.578} C_VEL
LIN {X 0,Y 440.692,Z 989.03,A -85,B 0,C 180,E1 8501.12,E2 8501.12} C_VEL
LIN {X 0,Y 440.735,Z 989.316,A -85,B 0,C 180,E1 8507.098,E2 8507.098} C_VEL
LIN {X 0,Y 445.467,Z 999.035,A -85,B 0,C 180,E1 8507.84,E2 8507.84} C_VEL
LIN {X 0,Y 467.236,Z 1040.26,A -85,B 0,C 180,E1 8510.904,E2 8510.904} C_VEL
LIN {X 0,Y 469.476,Z 1044.942,A -85,B 0,C 180,E1 8511.208,E2 8511.208} C_VEL
LIN {X 0,Y 467.004,Z 1087.7,A -85,B 0,C 180,E1 8512.294,E2 8512.294} C_VEL
LIN {X 0,Y 463.338,Z 1126.216,A -85,B 0,C 180,E1 8513.986,E2 8513.986} C_VEL
LIN {X 0,Y 458.759,Z 1163.845,A -85,B 0,C 180,E1 8516.409,E2 8516.409} C_VEL
LIN {X 0,Y 457.211,Z 1176.493,A -85,B 0,C 180,E1 8517.433,E2 8517.433} C_VEL
LIN {X 0,Y 451.592,Z 1190.859,A -85,B 0,C 180,E1 8518.519,E2 8518.519} C_VEL
LIN {X 0,Y 446.074,Z 1204.438,A -85,B 0,C 180,E1 8519.718,E2 8519.718} C_VEL
LIN {X 0,Y 441.602,Z 1236.611,A -85,B 0,C 180,E1 8523.799,E2 8523.799} C_VEL
LIN {X 0,Y 438.095,Z 1264.162,A -85,B 0,C 180,E1 8528.43,E2 8528.43} C_VEL
LIN {X 0,Y 435.94,Z 1284.232,A -85,B 0,C 180,E1 8532.888,E2 8532.888} C_VEL
LIN {X 0,Y 434.718,Z 1299.25,A -85,B 0,C 180,E1 8537.542,E2 8537.542} C_VEL
LIN {X 0,Y 434.207,Z 1308.216,A -85,B 0,C 180,E1 8542.009,E2 8542.009} C_VEL
LIN {X 0,Y 434.015,Z 1312.906,A -85,B 0,C 180,E1 8546.012,E2 8546.012} C_VEL
LIN {X 0,Y 434.045,Z 1314.5,A -85,B 0,C 180,E1 8549.999,E2 8549.999} C_VEL
LIN {X 0,Y 434.01,Z 1312.91,A -85,B 0,C 180,E1 8553.987,E2 8553.987} C_VEL
LIN {X 0,Y 434.288,Z 1306.599,A -85,B 0,C 180,E1 8558.995,E2 8558.995} C_VEL
LIN {X 0,Y 435.092,Z 1294.888,A -85,B 0,C 180,E1 8564.05,E2 8564.05} C_VEL
LIN {X 0,Y 436.677,Z 1276.884,A -85,B 0,C 180,E1 8568.902,E2 8568.902} C_VEL
LIN {X 0,Y 439.564,Z 1251.951,A -85,B 0,C 180,E1 8573.789,E2 8573.789} C_VEL
LIN {X 0,Y 443.395,Z 1223.532,A -85,B 0,C 180,E1 8577.995,E2 8577.995} C_VEL
LIN {X 0,Y 448.073,Z 1190.195,A -85,B 0,C 180,E1 8581.749,E2 8581.749} C_VEL
LIN {X 0,Y 453.088,Z 1153.861,A -85,B 0,C 180,E1 8584.796,E2 8584.796} C_VEL
LIN {X 0,Y 457.665,Z 1116.27,A -85,B 0,C 180,E1 8587.059,E2 8587.059} C_VEL
LIN {X 0,Y 461.414,Z 1078.435,A -85,B 0,C 180,E1 8588.565,E2 8588.565} C_VEL
LIN {X 0,Y 462.693,Z 1047.234,A -85,B 0,C 180,E1 8589.383,E2 8589.383} C_VEL
LIN {X 0,Y 443.419,Z 1009.236,A -85,B 0,C 180,E1 8592.179,E2 8592.179} C_VEL
LIN {X 0,Y 432.95,Z 990.554,A -85,B 0,C 180,E1 8593.803,E2 8593.803} C_VEL
LIN {X 0,Y 432.813,Z 989.03,A -85,B 0,C 180,E1 8593.953,E2 8593.953} C_VEL
LIN {X 0,Y 432.782,Z 989.03,A -85,B 0,C 180,E1 8600.092,E2 8600.092} C_VEL
LIN {X 0,Y 432.895,Z 989.03,A -85,B 0,C 180,E1 8606.782,E2 8606.782} C_VEL
LIN {X 0,Y 433.033,Z 989.03,A -85,B 0,C 180,E1 8613.064,E2 8613.064} C_VEL
LIN {X 0,Y 433.302,Z 989.03,A -85,B 0,C 180,E1 8620.1,E2 8620.1} C_VEL
LIN {X 0,Y 433.302,Z 989.03,A -85,B 0,C 180,E1 8625.891,E2 8625.891} C_VEL
LIN {X 0,Y 433.614,Z 989.03,A -85,B 0,C 180,E1 8631.999,E2 8631.999} C_VEL
LIN {X 0,Y 433.991,Z 989.03,A -85,B 0,C 180,E1 8638.007,E2 8638.007} C_VEL
LIN {X 0,Y 433.828,Z 989.03,A -85,B 0,C 180,E1 8643.989,E2 8643.989} C_VEL
LIN {X 0,Y 433.601,Z 989.03,A -85,B 0,C 180,E1 8650.021,E2 8650.021} C_VEL
LIN {X 0,Y 433.386,Z 989.03,A -85,B 0,C 180,E1 8656.173,E2 8656.173} C_VEL
LIN {X 0,Y 433.197,Z 989.03,A -85,B 0,C 180,E1 8662.53,E2 8662.53} C_VEL
LIN {X 0,Y 432.905,Z 989.03,A -85,B 0,C 180,E1 8669.374,E2 8669.374} C_VEL
LIN {X 0,Y 432.821,Z 989.03,A -85,B 0,C 180,E1 8673.904,E2 8673.904} C_VEL
LIN {X 0,Y 432.683,Z 989.03,A -85,B 0,C 180,E1 8679.892,E2 8679.892} C_VEL
LIN {X 0,Y 432.813,Z 989.03,A -85,B 0,C 180,E1 8687.066,E2 8687.066} C_VEL
LIN {X 0,Y 432.947,Z 989.463,A -85,B 0,C 180,E1 8690.136,E2 8690.136} C_VEL
LIN {X 0,Y 445.438,Z 1020.672,A -85,B 0,C 180,E1 8694.138,E2 8694.138} C_VEL
LIN {X 0,Y 451.594,Z 1045.272,A -85,B 0,C 180,E1 8697.332,E2 8697.332} C_VEL
LIN {X 0,Y 446.923,Z 1075.626,A -85,B 0,C 180,E1 8700.798,E2 8700.798} C_VEL
LIN {X 0,Y 441.973,Z 1102.706,A -85,B 0,C 180,E1 8704.913,E2 8704.913} C_VEL
LIN {X 0,Y 438.221,Z 1124.463,A -85,B 0,C 180,E1 8709.408,E2 8709.408} C_VEL
LIN {X 0,Y 435.672,Z 1141.936,A -85,B 0,C 180,E1 8714.43,E2 8714.43} C_VEL
LIN {X 0,Y 434.434,Z 1154.765,A -85,B 0,C 180,E1 8719.999,E2 8719.999} C_VEL
LIN {X 0,Y 434.084,Z 1161.013,A -85,B 0,C 180,E1 8724.014,E2 8724.014} C_VEL
LIN {X 0,Y 434.018,Z 1164.115,A -85,B 0,C 180,E1 8728.008,E2 8728.008} C_VEL
LIN {X 0,Y 434.083,Z 1164.067,A -85,B 0,C 180,E1 8731.993,E2 8731.993} C_VEL
LIN {X 0,Y 434.111,Z 1159.694,A -85,B 0,C 180,E1 8736.989,E2 8736.989} C_VEL
LIN {X 0,Y 434.921,Z 1148.527,A -85,B 0,C 180,E1 8742.933,E2 8742.933} C_VEL
LIN {X 0,Y 436.854,Z 1133.478,A -85,B 0,C 180,E1 8748.113,E2 8748.113} C_VEL
LIN {X 0,Y 440.112,Z 1113.346,A -85,B 0,C 180,E1 8752.956,E2 8752.956} C_VEL
LIN {X 0,Y 444.535,Z 1088.713,A -85,B 0,C 180,E1 8757.276,E2 8757.276} C_VEL
LIN {X 0,Y 449.927,Z 1058.506,A -85,B 0,C 180,E1 8761.172,E2 8761.172} C_VEL
LIN {X 0,Y 451.458,Z 1044.867,A -85,B 0,C 180,E1 8762.637,E2 8762.637} C_VEL
LIN {X 0,Y 445.711,Z 1021.539,A -85,B 0,C 180,E1 8765.658,E2 8765.658} C_VEL
LIN {X 0,Y 434.691,Z 994.068,A -85,B 0,C 180,E1 8769.226,E2 8769.226} C_VEL
LIN {X 0,Y 432.832,Z 989.03,A -85,B 0,C 180,E1 8769.918,E2 8769.918} C_VEL
LIN {X 0,Y 432.806,Z 989.03,A -85,B 0,C 180,E1 8777.071,E2 8777.071} C_VEL
LIN {X 0,Y 432.838,Z 989.03,A -85,B 0,C 180,E1 8783.655,E2 8783.655} C_VEL
LIN {X 0,Y 432.838,Z 989.03,A -85,B 0,C 180,E1 8788.471,E2 8788.471} C_VEL
LIN {X 0,Y 433.072,Z 989.03,A -85,B 0,C 180,E1 8795.284,E2 8795.284} C_VEL
LIN {X 0,Y 433.306,Z 989.03,A -85,B 0,C 180,E1 8801.735,E2 8801.735} C_VEL
LIN {X 0,Y 433.356,Z 989.03,A -85,B 0,C 180,E1 8807.941,E2 8807.941} C_VEL
LIN {X 0,Y 433.776,Z 989.03,A -85,B 0,C 180,E1 8814.01,E2 8814.01} C_VEL
LIN {X 0,Y 433.977,Z 989.03,A -85,B 0,C 180,E1 8820,E2 8820} C_VEL
LIN {X 0,Y 433.744,Z 989.03,A -85,B 0,C 180,E1 8825.991,E2 8825.991} C_VEL
LIN {X 0,Y 433.468,Z 989.03,A -85,B 0,C 180,E1 8832.899,E2 8832.899} C_VEL
LIN {X 0,Y 433.285,Z 989.03,A -85,B 0,C 180,E1 8838.266,E2 8838.266} C_VEL
LIN {X 0,Y 433.042,Z 989.03,A -85,B 0,C 180,E1 8845.038,E2 8845.038} C_VEL
LIN {X 0,Y 432.959,Z 989.03,A -85,B 0,C 180,E1 8851.519,E2 8851.519} C_VEL
LIN {X 0,Y 432.897,Z 989.03,A -85,B 0,C 180,E1 8856.702,E2 8856.702} C_VEL
LIN {X 0,Y 432.71,Z 989.03,A -85,B 0,C 180,E1 8862.916,E2 8862.916} C_VEL
LIN {X 0,Y 432.784,Z 989.03,A -85,B 0,C 180,E1 8866.127,E2 8866.127} C_VEL
LIN {X 0,Y 435.178,Z 994.698,A -85,B 0,C 180,E1 8866.562,E2 8866.562} C_VEL
LIN {X 0,Y 458.017,Z 1037.018,A -85,B 0,C 180,E1 8869.939,E2 8869.939} C_VEL
LIN {X 0,Y 463.104,Z 1048.951,A -85,B 0,C 180,E1 8870.696,E2 8870.696} C_VEL
LIN {X 0,Y 460.369,Z 1089.743,A -85,B 0,C 180,E1 8871.808,E2 8871.808} C_VEL
LIN {X 0,Y 456.518,Z 1126.649,A -85,B 0,C 180,E1 8873.487,E2 8873.487} C_VEL
LIN {X 0,Y 451.643,Z 1164.217,A -85,B 0,C 180,E1 8875.973,E2 8875.973} C_VEL
LIN {X 0,Y 446.821,Z 1199.082,A -85,B 0,C 180,E1 8879.152,E2 8879.152} C_VEL
LIN {X 0,Y 446.074,Z 1204.438,A -85,B 0,C 180,E1 8879.718,E2 8879.718} C_VEL
LIN {X 0,Y 440.434,Z 1217.431,A -85,B 0,C 180,E1 8881.059,E2 8881.059} C_VEL
LIN {X 0,Y 434.952,Z 1229.694,A -85,B 0,C 180,E1 8882.535,E2 8882.535} C_VEL
LIN {X 0,Y 431.143,Z 1257.785,A -85,B 0,C 180,E1 8887.083,E2 8887.083} C_VEL
LIN {X 0,Y 428.403,Z 1280.526,A -85,B 0,C 180,E1 8891.991,E2 8891.991} C_VEL
LIN {X 0,Y 426.943,Z 1297.19,A -85,B 0,C 180,E1 8896.96,E2 8896.96} C_VEL
LIN {X 0,Y 426.429,Z 1306.315,A -85,B 0,C 180,E1 8900.836,E2 8900.836} C_VEL
LIN {X 0,Y 426.176,Z 1310.926,A -85,B 0,C 180,E1 8903.902,E2 8903.902} C_VEL
LIN {X 0,Y 426.118,Z 1314.088,A -85,B 0,C 180,E1 8907.97,E2 8907.97} C_VEL
LIN {X 0,Y 426.157,Z 1314.09,A -85,B 0,C 180,E1 8912.029,E2 8912.029} C_VEL
LIN {X 0,Y 426.317,Z 1308.833,A -85,B 0,C 180,E1 8917.668,E2 8917.668} C_VEL
LIN {X 0,Y 426.937,Z 1298.312,A -85,B 0,C 180,E1 8922.648,E2 8922.648} C_VEL
LIN {X 0,Y 428.36,Z 1282.115,A -85,B 0,C 180,E1 8927.617,E2 8927.617} C_VEL
LIN {X 0,Y 430.886,Z 1259.202,A -85,B 0,C 180,E1 8932.657,E2 8932.657} C_VEL
LIN {X 0,Y 434.759,Z 1230.79,A -85,B 0,C 180,E1 8937.312,E2 8937.312} C_VEL
LIN {X 0,Y 439.538,Z 1198.743,A -85,B 0,C 180,E1 8941.282,E2 8941.282} C_VEL
LIN {X 0,Y 444.635,Z 1164.552,A -85,B 0,C 180,E1 8944.473,E2 8944.473} C_VEL
LIN {X 0,Y 449.537,Z 1128.525,A -85,B 0,C 180,E1 8946.946,E2 8946.946} C_VEL
LIN {X 0,Y 453.91,Z 1090.029,A -85,B 0,C 180,E1 8948.758,E2 8948.758} C_VEL
LIN {X 0,Y 456.703,Z 1050.625,A -85,B 0,C 180,E1 8949.892,E2 8949.892} C_VEL
LIN {X 0,Y 437.822,Z 1013.207,A -85,B 0,C 180,E1 8952.732,E2 8952.732} C_VEL
LIN {X 0,Y 424.929,Z 989.82,A -85,B 0,C 180,E1 8954.822,E2 8954.822} C_VEL
LIN {X 0,Y 424.881,Z 989.03,A -85,B 0,C 180,E1 8960.263,E2 8960.263} C_VEL
LIN {X 0,Y 424.866,Z 989.03,A -85,B 0,C 180,E1 8965.371,E2 8965.371} C_VEL
LIN {X 0,Y 424.953,Z 989.03,A -85,B 0,C 180,E1 8970.19,E2 8970.19} C_VEL
LIN {X 0,Y 425.268,Z 989.03,A -85,B 0,C 180,E1 8977.304,E2 8977.304} C_VEL
LIN {X 0,Y 425.343,Z 989.03,A -85,B 0,C 180,E1 8983.512,E2 8983.512} C_VEL
LIN {X 0,Y 425.522,Z 989.03,A -85,B 0,C 180,E1 8989.787,E2 8989.787} C_VEL
LIN {X 0,Y 425.863,Z 989.03,A -85,B 0,C 180,E1 8995.936,E2 8995.936} C_VEL
LIN {X 0,Y 425.93,Z 989.03,A -85,B 0,C 180,E1 9002.03,E2 9002.03} C_VEL
LIN {X 0,Y 425.708,Z 989.03,A -85,B 0,C 180,E1 9008.151,E2 9008.151} C_VEL
LIN {X 0,Y 425.522,Z 989.03,A -85,B 0,C 180,E1 9014.373,E2 9014.373} C_VEL
LIN {X 0,Y 425.29,Z 989.03,A -85,B 0,C 180,E1 9020.781,E2 9020.781} C_VEL
LIN {X 0,Y 425.047,Z 989.03,A -85,B 0,C 180,E1 9027.484,E2 9027.484} C_VEL
LIN {X 0,Y 424.903,Z 989.03,A -85,B 0,C 180,E1 9032.187,E2 9032.187} C_VEL
LIN {X 0,Y 424.766,Z 989.03,A -85,B 0,C 180,E1 9038.597,E2 9038.597} C_VEL
LIN {X 0,Y 424.858,Z 989.03,A -85,B 0,C 180,E1 9045.262,E2 9045.262} C_VEL
LIN {X 0,Y 424.95,Z 989.559,A -85,B 0,C 180,E1 9049.101,E2 9049.101} C_VEL
LIN {X 0,Y 437.543,Z 1019.926,A -85,B 0,C 180,E1 9053.146,E2 9053.146} C_VEL
LIN {X 0,Y 443.813,Z 1042.789,A -85,B 0,C 180,E1 9056.215,E2 9056.215} C_VEL
LIN {X 0,Y 444.668,Z 1051.648,A -85,B 0,C 180,E1 9057.338,E2 9057.338} C_VEL
LIN {X 0,Y 439.182,Z 1081.88,A -85,B 0,C 180,E1 9060.967,E2 9060.967} C_VEL
LIN {X 0,Y 434.294,Z 1107.096,A -85,B 0,C 180,E1 9065.036,E2 9065.036} C_VEL
LIN {X 0,Y 430.601,Z 1127.575,A -85,B 0,C 180,E1 9069.486,E2 9069.486} C_VEL
LIN {X 0,Y 427.926,Z 1144.704,A -85,B 0,C 180,E1 9074.665,E2 9074.665} C_VEL
LIN {X 0,Y 426.738,Z 1156.082,A -85,B 0,C 180,E1 9079.817,E2 9079.817} C_VEL
LIN {X 0,Y 426.244,Z 1161.67,A -85,B 0,C 180,E1 9083.904,E2 9083.904} C_VEL
LIN {X 0,Y 426.12,Z 1164.424,A -85,B 0,C 180,E1 9087.971,E2 9087.971} C_VEL
LIN {X 0,Y 426.184,Z 1164.37,A -85,B 0,C 180,E1 9092.03,E2 9092.03} C_VEL
LIN {X 0,Y 426.315,Z 1159.777,A -85,B 0,C 180,E1 9097.667,E2 9097.667} C_VEL
LIN {X 0,Y 427.246,Z 1150.208,A -85,B 0,C 180,E1 9103.043,E2 9103.043} C_VEL
LIN {X 0,Y 429.233,Z 1136.003,A -85,B 0,C 180,E1 9108.106,E2 9108.106} C_VEL
LIN {X 0,Y 432.425,Z 1117.185,A -85,B 0,C 180,E1 9112.845,E2 9112.845} C_VEL
LIN {X 0,Y 436.909,Z 1093.716,A -85,B 0,C 180,E1 9117.176,E2 9117.176} C_VEL
LIN {X 0,Y 442.041,Z 1066.306,A -85,B 0,C 180,E1 9120.951,E2 9120.951} C_VEL
LIN {X 0,Y 444.927,Z 1048.997,A -85,B 0,C 180,E1 9122.865,E2 9122.865} C_VEL
LIN {X 0,Y 439.298,Z 1025.249,A -85,B 0,C 180,E1 9126.037,E2 9126.037} C_VEL
LIN {X 0,Y 428.321,Z 997.753,A -85,B 0,C 180,E1 9129.766,E2 9129.766} C_VEL
LIN {X 0,Y 424.813,Z 989.03,A -85,B 0,C 180,E1 9130.958,E2 9130.958} C_VEL
LIN {X 0,Y 424.886,Z 989.03,A -85,B 0,C 180,E1 9137.564,E2 9137.564} C_VEL
LIN {X 0,Y 424.924,Z 989.03,A -85,B 0,C 180,E1 9142.866,E2 9142.866} C_VEL
LIN {X 0,Y 424.959,Z 989.03,A -85,B 0,C 180,E1 9150.191,E2 9150.191} C_VEL
LIN {X 0,Y 425.27,Z 989.03,A -85,B 0,C 180,E1 9157.307,E2 9157.307} C_VEL
LIN {X 0,Y 425.361,Z 989.03,A -85,B 0,C 180,E1 9163.513,E2 9163.513} C_VEL
LIN {X 0,Y 425.567,Z 989.03,A -85,B 0,C 180,E1 9169.788,E2 9169.788} C_VEL
LIN {X 0,Y 425.874,Z 989.03,A -85,B 0,C 180,E1 9175.936,E2 9175.936} C_VEL
LIN {X 0,Y 425.921,Z 989.03,A -85,B 0,C 180,E1 9182.03,E2 9182.03} C_VEL
LIN {X 0,Y 425.717,Z 989.03,A -85,B 0,C 180,E1 9188.151,E2 9188.151} C_VEL
LIN {X 0,Y 425.53,Z 989.03,A -85,B 0,C 180,E1 9194.372,E2 9194.372} C_VEL
LIN {X 0,Y 425.287,Z 989.03,A -85,B 0,C 180,E1 9200.782,E2 9200.782} C_VEL
LIN {X 0,Y 425.084,Z 989.03,A -85,B 0,C 180,E1 9207.482,E2 9207.482} C_VEL
LIN {X 0,Y 425.035,Z 989.03,A -85,B 0,C 180,E1 9212.176,E2 9212.176} C_VEL
LIN {X 0,Y 424.909,Z 989.03,A -85,B 0,C 180,E1 9218.619,E2 9218.619} C_VEL
LIN {X 0,Y 424.818,Z 989.03,A -85,B 0,C 180,E1 9225.114,E2 9225.114} C_VEL
LIN {X 0,Y 427.414,Z 994.856,A -85,B 0,C 180,E1 9225.615,E2 9225.615} C_VEL
LIN {X 0,Y 450.855,Z 1037.849,A -85,B 0,C 180,E1 9229.22,E2 9229.22} C_VEL
LIN {X 0,Y 456.825,Z 1051.618,A -85,B 0,C 180,E1 9230.145,E2 9230.145} C_VEL
LIN {X 0,Y 453.564,Z 1093.54,A -85,B 0,C 180,E1 9231.368,E2 9231.368} C_VEL
LIN {X 0,Y 448.928,Z 1133.847,A -85,B 0,C 180,E1 9233.366,E2 9233.366} C_VEL
LIN {X 0,Y 443.495,Z 1172.223,A -85,B 0,C 180,E1 9236.158,E2 9236.158} C_VEL
LIN {X 0,Y 438.324,Z 1206.597,A -85,B 0,C 180,E1 9239.587,E2 9239.587} C_VEL
LIN {X 0,Y 434.952,Z 1229.694,A -85,B 0,C 180,E1 9242.535,E2 9242.535} C_VEL
LIN {X 0,Y 432.906,Z 1235.615,A -85,B 0,C 180,E1 9243.345,E2 9243.345} C_VEL
LIN {X 0,Y 424.258,Z 1250.732,A -85,B 0,C 180,E1 9245.603,E2 9245.603} C_VEL
LIN {X 0,Y 424.009,Z 1252.016,A -85,B 0,C 180,E1 9245.84,E2 9245.84} C_VEL
LIN {X 0,Y 421.009,Z 1276.134,A -85,B 0,C 180,E1 9250.908,E2 9250.908} C_VEL
LIN {X 0,Y 419.323,Z 1293.75,A -85,B 0,C 180,E1 9255.988,E2 9255.988} C_VEL
LIN {X 0,Y 418.609,Z 1304.937,A -85,B 0,C 180,E1 9260.664,E2 9260.664} C_VEL
LIN {X 0,Y 418.266,Z 1311.985,A -85,B 0,C 180,E1 9265.861,E2 9265.861} C_VEL
LIN {X 0,Y 418.277,Z 1313.777,A -85,B 0,C 180,E1 9269.999,E2 9269.999} C_VEL
LIN {X 0,Y 418.252,Z 1311.021,A -85,B 0,C 180,E1 9275.174,E2 9275.174} C_VEL
LIN {X 0,Y 418.611,Z 1303.871,A -85,B 0,C 180,E1 9279.858,E2 9279.858} C_VEL
LIN {X 0,Y 419.441,Z 1292.105,A -85,B 0,C 180,E1 9284.586,E2 9284.586} C_VEL
LIN {X 0,Y 421.365,Z 1272.828,A -85,B 0,C 180,E1 9289.889,E2 9289.889} C_VEL
LIN {X 0,Y 424.401,Z 1249.016,A -85,B 0,C 180,E1 9294.694,E2 9294.694} C_VEL
LIN {X 0,Y 428.78,Z 1220.083,A -85,B 0,C 180,E1 9299.109,E2 9299.109} C_VEL
LIN {X 0,Y 433.972,Z 1187.251,A -85,B 0,C 180,E1 9302.909,E2 9302.909} C_VEL
LIN {X 0,Y 439.611,Z 1151.399,A -85,B 0,C 180,E1 9305.988,E2 9305.988} C_VEL
LIN {X 0,Y 444.736,Z 1113.847,A -85,B 0,C 180,E1 9308.3,E2 9308.3} C_VEL
LIN {X 0,Y 449.087,Z 1074.761,A -85,B 0,C 180,E1 9309.864,E2 9309.864} C_VEL
LIN {X 0,Y 450.055,Z 1052.418,A -85,B 0,C 180,E1 9310.524,E2 9310.524} C_VEL
LIN {X 0,Y 431.326,Z 1015.284,A -85,B 0,C 180,E1 9313.455,E2 9313.455} C_VEL
LIN {X 0,Y 417.091,Z 990.619,A -85,B 0,C 180,E1 9315.837,E2 9315.837} C_VEL
LIN {X 0,Y 416.931,Z 989.03,A -85,B 0,C 180,E1 9316.028,E2 9316.028} C_VEL
LIN {X 0,Y 417.027,Z 989.03,A -85,B 0,C 180,E1 9322.755,E2 9322.755} C_VEL
LIN {X 0,Y 417.057,Z 989.03,A -85,B 0,C 180,E1 9330.269,E2 9330.269} C_VEL
LIN {X 0,Y 417.251,Z 989.03,A -85,B 0,C 180,E1 9336.559,E2 9336.559} C_VEL
LIN {X 0,Y 417.431,Z 989.03,A -85,B 0,C 180,E1 9343.191,E2 9343.191} C_VEL
LIN {X 0,Y 417.591,Z 989.03,A -85,B 0,C 180,E1 9349.591,E2 9349.591} C_VEL
LIN {X 0,Y 417.951,Z 989.03,A -85,B 0,C 180,E1 9355.859,E2 9355.859} C_VEL
LIN {X 0,Y 418.054,Z 989.03,A -85,B 0,C 180,E1 9362.068,E2 9362.068} C_VEL
LIN {X 0,Y 417.785,Z 989.03,A -85,B 0,C 180,E1 9368.307,E2 9368.307} C_VEL
LIN {X 0,Y 417.592,Z 989.03,A -85,B 0,C 180,E1 9374.652,E2 9374.652} C_VEL
LIN {X 0,Y 417.358,Z 989.03,A -85,B 0,C 180,E1 9381.195,E2 9381.195} C_VEL
LIN {X 0,Y 417.058,Z 989.03,A -85,B 0,C 180,E1 9388.057,E2 9388.057} C_VEL
LIN {X 0,Y 416.87,Z 989.03,A -85,B 0,C 180,E1 9395.391,E2 9395.391} C_VEL
LIN {X 0,Y 416.824,Z 989.03,A -85,B 0,C 180,E1 9400.664,E2 9400.664} C_VEL
LIN {X 0,Y 417.044,Z 989.718,A -85,B 0,C 180,E1 9408.026,E2 9408.026} C_VEL
LIN {X 0,Y 430.268,Z 1020.895,A -85,B 0,C 180,E1 9412.356,E2 9412.356} C_VEL
LIN {X 0,Y 437.037,Z 1045.167,A -85,B 0,C 180,E1 9415.729,E2 9415.729} C_VEL
LIN {X 0,Y 437.904,Z 1054.111,A -85,B 0,C 180,E1 9416.903,E2 9416.903} C_VEL
LIN {X 0,Y 432.355,Z 1083.254,A -85,B 0,C 180,E1 9420.463,E2 9420.463} C_VEL
LIN {X 0,Y 427.179,Z 1108.478,A -85,B 0,C 180,E1 9424.591,E2 9424.591} C_VEL
LIN {X 0,Y 423.245,Z 1128.96,A -85,B 0,C 180,E1 9429.113,E2 9429.113} C_VEL
LIN {X 0,Y 420.367,Z 1146.087,A -85,B 0,C 180,E1 9434.382,E2 9434.382} C_VEL
LIN {X 0,Y 419.048,Z 1157.46,A -85,B 0,C 180,E1 9439.628,E2 9439.628} C_VEL
LIN {X 0,Y 418.486,Z 1163.046,A -85,B 0,C 180,E1 9443.791,E2 9443.791} C_VEL
LIN {X 0,Y 418.354,Z 1165.795,A -85,B 0,C 180,E1 9447.934,E2 9447.934} C_VEL
LIN {X 0,Y 418.411,Z 1165.743,A -85,B 0,C 180,E1 9452.068,E2 9452.068} C_VEL
LIN {X 0,Y 418.558,Z 1161.656,A -85,B 0,C 180,E1 9457.434,E2 9457.434} C_VEL
LIN {X 0,Y 419.378,Z 1153.4,A -85,B 0,C 180,E1 9462.469,E2 9462.469} C_VEL
LIN {X 0,Y 421.558,Z 1138.876,A -85,B 0,C 180,E1 9467.994,E2 9467.994} C_VEL
LIN {X 0,Y 424.983,Z 1119.794,A -85,B 0,C 180,E1 9472.992,E2 9472.992} C_VEL
LIN {X 0,Y 429.693,Z 1096.485,A -85,B 0,C 180,E1 9477.431,E2 9477.431} C_VEL
LIN {X 0,Y 435.155,Z 1068.825,A -85,B 0,C 180,E1 9481.344,E2 9481.344} C_VEL
LIN {X 0,Y 437.941,Z 1050.476,A -85,B 0,C 180,E1 9483.458,E2 9483.458} C_VEL
LIN {X 0,Y 432.937,Z 1029.055,A -85,B 0,C 180,E1 9486.415,E2 9486.415} C_VEL
LIN {X 0,Y 421.741,Z 999.893,A -85,B 0,C 180,E1 9490.469,E2 9490.469} C_VEL
LIN {X 0,Y 416.904,Z 989.03,A -85,B 0,C 180,E1 9491.971,E2 9491.971} C_VEL
LIN {X 0,Y 416.931,Z 989.03,A -85,B 0,C 180,E1 9499.349,E2 9499.349} C_VEL
LIN {X 0,Y 416.966,Z 989.03,A -85,B 0,C 180,E1 9504.619,E2 9504.619} C_VEL
LIN {X 0,Y 417.066,Z 989.03,A -85,B 0,C 180,E1 9511.944,E2 9511.944} C_VEL
LIN {X 0,Y 417.372,Z 989.03,A -85,B 0,C 180,E1 9518.806,E2 9518.806} C_VEL
LIN {X 0,Y 417.441,Z 989.03,A -85,B 0,C 180,E1 9525.343,E2 9525.343} C_VEL
LIN {X 0,Y 417.799,Z 989.03,A -85,B 0,C 180,E1 9531.694,E2 9531.694} C_VEL
LIN {X 0,Y 418.202,Z 989.03,A -85,B 0,C 180,E1 9537.932,E2 9537.932} C_VEL
LIN {X 0,Y 418.014,Z 989.03,A -85,B 0,C 180,E1 9544.14,E2 9544.14} C_VEL
LIN {X 0,Y 417.749,Z 989.03,A -85,B 0,C 180,E1 9550.405,E2 9550.405} C_VEL
LIN {X 0,Y 417.505,Z 989.03,A -85,B 0,C 180,E1 9556.806,E2 9556.806} C_VEL
LIN {X 0,Y 417.255,Z 989.03,A -85,B 0,C 180,E1 9563.441,E2 9563.441} C_VEL
LIN {X 0,Y 417.11,Z 989.03,A -85,B 0,C 180,E1 9570.429,E2 9570.429} C_VEL
LIN {X 0,Y 417.064,Z 989.03,A -85,B 0,C 180,E1 9577.249,E2 9577.249} C_VEL
LIN {X 0,Y 416.859,Z 989.03,A -85,B 0,C 180,E1 9584.102,E2 9584.102} C_VEL
LIN {X 0,Y 419.27,Z 994.663,A -85,B 0,C 180,E1 9584.559,E2 9584.559} C_VEL
LIN {X 0,Y 442.037,Z 1035.231,A -85,B 0,C 180,E1 9588.216,E2 9588.216} C_VEL
LIN {X 0,Y 450.466,Z 1054.542,A -85,B 0,C 180,E1 9589.582,E2 9589.582} C_VEL
LIN {X 0,Y 446.916,Z 1095.556,A -85,B 0,C 180,E1 9590.866,E2 9590.866} C_VEL
LIN {X 0,Y 442.238,Z 1133.544,A -85,B 0,C 180,E1 9592.808,E2 9592.808} C_VEL
LIN {X 0,Y 436.692,Z 1170.586,A -85,B 0,C 180,E1 9595.539,E2 9595.539} C_VEL
LIN {X 0,Y 431.099,Z 1205.588,A -85,B 0,C 180,E1 9599.082,E2 9599.082} C_VEL
LIN {X 0,Y 426.351,Z 1236.006,A -85,B 0,C 180,E1 9603.174,E2 9603.174} C_VEL
LIN {X 0,Y 424.009,Z 1252.016,A -85,B 0,C 180,E1 9605.84,E2 9605.84} C_VEL
LIN {X 0,Y 420.534,Z 1259.623,A -85,B 0,C 180,E1 9607.232,E2 9607.232} C_VEL
LIN {X 0,Y 413.908,Z 1269.857,A -85,B 0,C 180,E1 9609.372,E2 9609.372} C_VEL
LIN {X 0,Y 413.707,Z 1270.973,A -85,B 0,C 180,E1 9609.63,E2 9609.63} C_VEL
LIN {X 0,Y 411.644,Z 1290.676,A -85,B 0,C 180,E1 9615.13,E2 9615.13} C_VEL
LIN {X 0,Y 410.798,Z 1303.54,A -85,B 0,C 180,E1 9620.484,E2 9620.484} C_VEL
LIN {X 0,Y 410.476,Z 1310.607,A -85,B 0,C 180,E1 9625.783,E2 9625.783} C_VEL
LIN {X 0,Y 410.519,Z 1312.408,A -85,B 0,C 180,E1 9629.999,E2 9629.999} C_VEL
LIN {X 0,Y 410.481,Z 1309.644,A -85,B 0,C 180,E1 9635.272,E2 9635.272} C_VEL
LIN {X 0,Y 410.873,Z 1301.404,A -85,B 0,C 180,E1 9640.581,E2 9640.581} C_VEL
LIN {X 0,Y 411.789,Z 1289,A -85,B 0,C 180,E1 9645.407,E2 9645.407} C_VEL
LIN {X 0,Y 413.754,Z 1270.193,A -85,B 0,C 180,E1 9650.55,E2 9650.55} C_VEL
LIN {X 0,Y 417.209,Z 1245.427,A -85,B 0,C 180,E1 9655.539,E2 9655.539} C_VEL
LIN {X 0,Y 421.746,Z 1217.048,A -85,B 0,C 180,E1 9659.869,E2 9659.869} C_VEL
LIN {X 0,Y 427.301,Z 1184.251,A -85,B 0,C 180,E1 9663.666,E2 9663.666} C_VEL
LIN {X 0,Y 433.223,Z 1148.132,A -85,B 0,C 180,E1 9666.764,E2 9666.764} C_VEL
LIN {X 0,Y 438.595,Z 1110.625,A -85,B 0,C 180,E1 9669.05,E2 9669.05} C_VEL
LIN {X 0,Y 443.165,Z 1071.315,A -85,B 0,C 180,E1 9670.589,E2 9670.589} C_VEL
LIN {X 0,Y 443.775,Z 1055.305,A -85,B 0,C 180,E1 9671.085,E2 9671.085} C_VEL
LIN {X 0,Y 426.08,Z 1019.73,A -85,B 0,C 180,E1 9673.998,E2 9673.998} C_VEL
LIN {X 0,Y 409.006,Z 989.797,A -85,B 0,C 180,E1 9676.986,E2 9676.986} C_VEL
LIN {X 0,Y 409.045,Z 989.03,A -85,B 0,C 180,E1 9683.827,E2 9683.827} C_VEL
LIN {X 0,Y 409.119,Z 989.03,A -85,B 0,C 180,E1 9691.349,E2 9691.349} C_VEL
LIN {X 0,Y 409.39,Z 989.03,A -85,B 0,C 180,E1 9698.372,E2 9698.372} C_VEL
LIN {X 0,Y 409.497,Z 989.03,A -85,B 0,C 180,E1 9705.052,E2 9705.052} C_VEL
LIN {X 0,Y 409.816,Z 989.03,A -85,B 0,C 180,E1 9711.531,E2 9711.531} C_VEL
LIN {X 0,Y 410.276,Z 989.03,A -85,B 0,C 180,E1 9717.892,E2 9717.892} C_VEL
LIN {X 0,Y 410.081,Z 989.03,A -85,B 0,C 180,E1 9724.22,E2 9724.22} C_VEL
LIN {X 0,Y 409.825,Z 989.03,A -85,B 0,C 180,E1 9730.608,E2 9730.608} C_VEL
LIN {X 0,Y 409.562,Z 989.03,A -85,B 0,C 180,E1 9737.142,E2 9737.142} C_VEL
LIN {X 0,Y 409.307,Z 989.03,A -85,B 0,C 180,E1 9743.924,E2 9743.924} C_VEL
LIN {X 0,Y 409.016,Z 989.03,A -85,B 0,C 180,E1 9751.097,E2 9751.097} C_VEL
LIN {X 0,Y 408.951,Z 989.03,A -85,B 0,C 180,E1 9756.183,E2 9756.183} C_VEL
LIN {X 0,Y 408.823,Z 989.03,A -85,B 0,C 180,E1 9762.421,E2 9762.421} C_VEL
LIN {X 0,Y 409.046,Z 989.393,A -85,B 0,C 180,E1 9766.856,E2 9766.856} C_VEL
LIN {X 0,Y 422.66,Z 1021.015,A -85,B 0,C 180,E1 9771.41,E2 9771.41} C_VEL
LIN {X 0,Y 430.137,Z 1046.679,A -85,B 0,C 180,E1 9775.105,E2 9775.105} C_VEL
LIN {X 0,Y 431.174,Z 1056.689,A -85,B 0,C 180,E1 9776.47,E2 9776.47} C_VEL
LIN {X 0,Y 425.181,Z 1086.429,A -85,B 0,C 180,E1 9780.207,E2 9780.207} C_VEL
LIN {X 0,Y 419.784,Z 1111.44,A -85,B 0,C 180,E1 9784.446,E2 9784.446} C_VEL
LIN {X 0,Y 415.532,Z 1132.324,A -85,B 0,C 180,E1 9789.264,E2 9789.264} C_VEL
LIN {X 0,Y 412.579,Z 1148.857,A -85,B 0,C 180,E1 9794.624,E2 9794.624} C_VEL
LIN {X 0,Y 411.341,Z 1158.843,A -85,B 0,C 180,E1 9799.431,E2 9799.431} C_VEL
LIN {X 0,Y 410.732,Z 1164.422,A -85,B 0,C 180,E1 9803.673,E2 9803.673} C_VEL
LIN {X 0,Y 410.59,Z 1167.165,A -85,B 0,C 180,E1 9807.895,E2 9807.895} C_VEL
LIN {X 0,Y 410.646,Z 1167.114,A -85,B 0,C 180,E1 9812.107,E2 9812.107} C_VEL
LIN {X 0,Y 410.798,Z 1163.297,A -85,B 0,C 180,E1 9817.358,E2 9817.358} C_VEL
LIN {X 0,Y 411.739,Z 1154.783,A -85,B 0,C 180,E1 9822.704,E2 9822.704} C_VEL
LIN {X 0,Y 414.142,Z 1139.918,A -85,B 0,C 180,E1 9828.435,E2 9828.435} C_VEL
LIN {X 0,Y 417.988,Z 1119.964,A -85,B 0,C 180,E1 9833.681,E2 9833.681} C_VEL
LIN {X 0,Y 423.241,Z 1095.536,A -85,B 0,C 180,E1 9838.299,E2 9838.299} C_VEL
LIN {X 0,Y 429.124,Z 1067.253,A -85,B 0,C 180,E1 9842.238,E2 9842.238} C_VEL
LIN {X 0,Y 431.284,Z 1053.878,A -85,B 0,C 180,E1 9843.793,E2 9843.793} C_VEL
LIN {X 0,Y 426.726,Z 1033.269,A -85,B 0,C 180,E1 9846.742,E2 9846.742} C_VEL
LIN {X 0,Y 416.374,Z 1005.641,A -85,B 0,C 180,E1 9850.72,E2 9850.72} C_VEL
LIN {X 0,Y 408.961,Z 989.03,A -85,B 0,C 180,E1 9853.121,E2 9853.121} C_VEL
LIN {X 0,Y 408.905,Z 989.03,A -85,B 0,C 180,E1 9858.376,E2 9858.376} C_VEL
LIN {X 0,Y 409.072,Z 989.03,A -85,B 0,C 180,E1 9864.249,E2 9864.249} C_VEL
LIN {X 0,Y 409.128,Z 989.03,A -85,B 0,C 180,E1 9871.35,E2 9871.35} C_VEL
LIN {X 0,Y 409.4,Z 989.03,A -85,B 0,C 180,E1 9878.372,E2 9878.372} C_VEL
LIN {X 0,Y 409.508,Z 989.03,A -85,B 0,C 180,E1 9885.053,E2 9885.053} C_VEL
LIN {X 0,Y 409.896,Z 989.03,A -85,B 0,C 180,E1 9891.532,E2 9891.532} C_VEL
LIN {X 0,Y 410.288,Z 989.03,A -85,B 0,C 180,E1 9897.892,E2 9897.892} C_VEL
LIN {X 0,Y 410.098,Z 989.03,A -85,B 0,C 180,E1 9904.22,E2 9904.22} C_VEL
LIN {X 0,Y 409.835,Z 989.03,A -85,B 0,C 180,E1 9910.608,E2 9910.608} C_VEL
LIN {X 0,Y 409.563,Z 989.03,A -85,B 0,C 180,E1 9917.142,E2 9917.142} C_VEL
LIN {X 0,Y 409.313,Z 989.03,A -85,B 0,C 180,E1 9923.924,E2 9923.924} C_VEL
LIN {X 0,Y 409.117,Z 989.03,A -85,B 0,C 180,E1 9931.089,E2 9931.089} C_VEL
LIN {X 0,Y 409.103,Z 989.03,A -85,B 0,C 180,E1 9936.168,E2 9936.168} C_VEL
LIN {X 0,Y 408.928,Z 989.728,A -85,B 0,C 180,E1 9943.012,E2 9943.012} C_VEL
LIN {X 0,Y 411.902,Z 995.168,A -85,B 0,C 180,E1 9943.566,E2 9943.566} C_VEL
LIN {X 0,Y 436.218,Z 1038.616,A -85,B 0,C 180,E1 9947.64,E2 9947.64} C_VEL
LIN {X 0,Y 444.149,Z 1056.649,A -85,B 0,C 180,E1 9948.999,E2 9948.999} C_VEL
LIN {X 0,Y 440.454,Z 1095.999,A -85,B 0,C 180,E1 9950.283,E2 9950.283} C_VEL
LIN {X 0,Y 435.502,Z 1133.745,A -85,B 0,C 180,E1 9952.265,E2 9952.265} C_VEL
LIN {X 0,Y 429.671,Z 1170.565,A -85,B 0,C 180,E1 9955.047,E2 9955.047} C_VEL
LIN {X 0,Y 423.827,Z 1205.07,A -85,B 0,C 180,E1 9958.62,E2 9958.62} C_VEL
LIN {X 0,Y 418.929,Z 1234.536,A -85,B 0,C 180,E1 9962.66,E2 9962.66} C_VEL
LIN {X 0,Y 414.922,Z 1261.352,A -85,B 0,C 180,E1 9967.498,E2 9967.498} C_VEL
LIN {X 0,Y 413.707,Z 1270.973,A -85,B 0,C 180,E1 9969.63,E2 9969.63} C_VEL
LIN {X 0,Y 410.514,Z 1277.233,A -85,B 0,C 180,E1 9971.172,E2 9971.172} C_VEL
LIN {X 0,Y 404.25,Z 1285.37,A -85,B 0,C 180,E1 9973.569,E2 9973.569} C_VEL
LIN {X 0,Y 404.079,Z 1286.233,A -85,B 0,C 180,E1 9973.854,E2 9973.854} C_VEL
LIN {X 0,Y 403.143,Z 1300.013,A -85,B 0,C 180,E1 9979.212,E2 9979.212} C_VEL
LIN {X 0,Y 402.815,Z 1307.045,A -85,B 0,C 180,E1 9983.546,E2 9983.546} C_VEL
LIN {X 0,Y 402.692,Z 1310.564,A -85,B 0,C 180,E1 9987.852,E2 9987.852} C_VEL
LIN {X 0,Y 402.727,Z 1310.572,A -85,B 0,C 180,E1 9992.147,E2 9992.147} C_VEL
LIN {X 0,Y 402.811,Z 1305.962,A -85,B 0,C 180,E1 9997.313,E2 9997.313} C_VEL
LIN {X 0,Y 403.335,Z 1296.404,A -85,B 0,C 180,E1 10002.422,E2 10002.422} C_VEL
LIN {X 0,Y 404.573,Z 1282.318,A -85,B 0,C 180,E1 10007.36,E2 10007.36} C_VEL
LIN {X 0,Y 407.093,Z 1261.337,A -85,B 0,C 180,E1 10012.638,E2 10012.638} C_VEL
LIN {X 0,Y 411.278,Z 1234.786,A -85,B 0,C 180,E1 10017.594,E2 10017.594} C_VEL
LIN {X 0,Y 416.619,Z 1204.485,A -85,B 0,C 180,E1 10021.866,E2 10021.866} C_VEL
LIN {X 0,Y 422.441,Z 1172.031,A -85,B 0,C 180,E1 10025.326,E2 10025.326} C_VEL
LIN {X 0,Y 428.438,Z 1135.437,A -85,B 0,C 180,E1 10028.211,E2 10028.211} C_VEL
LIN {X 0,Y 433.998,Z 1096.729,A -85,B 0,C 180,E1 10030.306,E2 10030.306} C_VEL
LIN {X 0,Y 437.497,Z 1057.904,A -85,B 0,C 180,E1 10031.673,E2 10031.673} C_VEL
LIN {X 0,Y 419.403,Z 1021.386,A -85,B 0,C 180,E1 10034.81,E2 10034.81} C_VEL
LIN {X 0,Y 402.362,Z 993.459,A -85,B 0,C 180,E1 10037.873,E2 10037.873} C_VEL
LIN {X 0,Y 401.027,Z 989.03,A -85,B 0,C 180,E1 10038.332,E2 10038.332} C_VEL
LIN {X 0,Y 401.089,Z 989.03,A -85,B 0,C 180,E1 10045.645,E2 10045.645} C_VEL
LIN {X 0,Y 401.253,Z 989.03,A -85,B 0,C 180,E1 10053.175,E2 10053.175} C_VEL
LIN {X 0,Y 401.512,Z 989.03,A -85,B 0,C 180,E1 10060.231,E2 10060.231} C_VEL
LIN {X 0,Y 401.699,Z 989.03,A -85,B 0,C 180,E1 10067.606,E2 10067.606} C_VEL
LIN {X 0,Y 402.116,Z 989.03,A -85,B 0,C 180,E1 10073.536,E2 10073.536} C_VEL
LIN {X 0,Y 402.328,Z 989.03,A -85,B 0,C 180,E1 10080,E2 10080} C_VEL
LIN {X 0,Y 402.087,Z 989.03,A -85,B 0,C 180,E1 10086.464,E2 10086.464} C_VEL
LIN {X 0,Y 401.835,Z 989.03,A -85,B 0,C 180,E1 10093.021,E2 10093.021} C_VEL
LIN {X 0,Y 401.491,Z 989.03,A -85,B 0,C 180,E1 10100.013,E2 10100.013} C_VEL
LIN {X 0,Y 401.244,Z 989.03,A -85,B 0,C 180,E1 10106.826,E2 10106.826} C_VEL
LIN {X 0,Y 401.02,Z 989.03,A -85,B 0,C 180,E1 10114.362,E2 10114.362} C_VEL
LIN {X 0,Y 400.875,Z 989.03,A -85,B 0,C 180,E1 10121.163,E2 10121.163} C_VEL
LIN {X 0,Y 401.015,Z 989.469,A -85,B 0,C 180,E1 10125.638,E2 10125.638} C_VEL
LIN {X 0,Y 414.367,Z 1019.244,A -85,B 0,C 180,E1 10130.138,E2 10130.138} C_VEL
LIN {X 0,Y 422.718,Z 1045.585,A -85,B 0,C 180,E1 10134.066,E2 10134.066} C_VEL
LIN {X 0,Y 424.508,Z 1059.01,A -85,B 0,C 180,E1 10135.993,E2 10135.993} C_VEL
LIN {X 0,Y 418.407,Z 1087.807,A -85,B 0,C 180,E1 10139.675,E2 10139.675} C_VEL
LIN {X 0,Y 412.704,Z 1112.824,A -85,B 0,C 180,E1 10143.976,E2 10143.976} C_VEL
LIN {X 0,Y 408.167,Z 1133.71,A -85,B 0,C 180,E1 10148.872,E2 10148.872} C_VEL
LIN {X 0,Y 405.025,Z 1150.237,A -85,B 0,C 180,E1 10154.33,E2 10154.33} C_VEL
LIN {X 0,Y 403.654,Z 1160.222,A -85,B 0,C 180,E1 10159.228,E2 10159.228} C_VEL
LIN {X 0,Y 403.002,Z 1165.794,A -85,B 0,C 180,E1 10163.551,E2 10163.551} C_VEL
LIN {X 0,Y 402.827,Z 1168.536,A -85,B 0,C 180,E1 10167.854,E2 10167.854} C_VEL
LIN {X 0,Y 402.878,Z 1168.486,A -85,B 0,C 180,E1 10172.147,E2 10172.147} C_VEL
LIN {X 0,Y 403.074,Z 1164.672,A -85,B 0,C 180,E1 10177.5,E2 10177.5} C_VEL
LIN {X 0,Y 404.095,Z 1156.168,A -85,B 0,C 180,E1 10182.948,E2 10182.948} C_VEL
LIN {X 0,Y 406.679,Z 1141.309,A -85,B 0,C 180,E1 10188.786,E2 10188.786} C_VEL
LIN {X 0,Y 410.808,Z 1121.353,A -85,B 0,C 180,E1 10194.121,E2 10194.121} C_VEL
LIN {X 0,Y 416.099,Z 1098.084,A -85,B 0,C 180,E1 10198.619,E2 10198.619} C_VEL
LIN {X 0,Y 422.239,Z 1070.108,A -85,B 0,C 180,E1 10202.623,E2 10202.623} C_VEL
LIN {X 0,Y 424.457,Z 1056.239,A -85,B 0,C 180,E1 10204.291,E2 10204.291} C_VEL
LIN {X 0,Y 419.987,Z 1035.806,A -85,B 0,C 180,E1 10207.311,E2 10207.311} C_VEL
LIN {X 0,Y 410.323,Z 1009.767,A -85,B 0,C 180,E1 10211.213,E2 10211.213} C_VEL
LIN {X 0,Y 401.006,Z 989.797,A -85,B 0,C 180,E1 10214.239,E2 10214.239} C_VEL
LIN {X 0,Y 401.016,Z 989.03,A -85,B 0,C 180,E1 10220.232,E2 10220.232} C_VEL
LIN {X 0,Y 401.089,Z 989.03,A -85,B 0,C 180,E1 10225.865,E2 10225.865} C_VEL
LIN {X 0,Y 401.246,Z 989.03,A -85,B 0,C 180,E1 10233.174,E2 10233.174} C_VEL
LIN {X 0,Y 401.534,Z 989.03,A -85,B 0,C 180,E1 10240.232,E2 10240.232} C_VEL
LIN {X 0,Y 401.721,Z 989.03,A -85,B 0,C 180,E1 10247.599,E2 10247.599} C_VEL
LIN {X 0,Y 402.151,Z 989.03,A -85,B 0,C 180,E1 10253.537,E2 10253.537} C_VEL
LIN {X 0,Y 402.39,Z 989.03,A -85,B 0,C 180,E1 10260,E2 10260} C_VEL
LIN {X 0,Y 402.098,Z 989.03,A -85,B 0,C 180,E1 10266.464,E2 10266.464} C_VEL
LIN {X 0,Y 401.847,Z 989.03,A -85,B 0,C 180,E1 10273.021,E2 10273.021} C_VEL
LIN {X 0,Y 401.483,Z 989.03,A -85,B 0,C 180,E1 10280.005,E2 10280.005} C_VEL
LIN {X 0,Y 401.279,Z 989.03,A -85,B 0,C 180,E1 10286.823,E2 10286.823} C_VEL
LIN {X 0,Y 401.183,Z 989.03,A -85,B 0,C 180,E1 10294.346,E2 10294.346} C_VEL
LIN {X 0,Y 400.99,Z 989.03,A -85,B 0,C 180,E1 10301.665,E2 10301.665} C_VEL
LIN {X 0,Y 401.038,Z 990.064,A -85,B 0,C 180,E1 10301.852,E2 10301.852} C_VEL
LIN {X 0,Y 427.032,Z 1035.523,A -85,B 0,C 180,E1 10306.484,E2 10306.484} C_VEL
LIN {X 0,Y 437.804,Z 1059.524,A -85,B 0,C 180,E1 10308.417,E2 10308.417} C_VEL
LIN {X 0,Y 433.593,Z 1100.078,A -85,B 0,C 180,E1 10309.842,E2 10309.842} C_VEL
LIN {X 0,Y 428.077,Z 1138.606,A -85,B 0,C 180,E1 10312.01,E2 10312.01} C_VEL
LIN {X 0,Y 421.665,Z 1176.349,A -85,B 0,C 180,E1 10315.068,E2 10315.068} C_VEL
LIN {X 0,Y 415.384,Z 1211.214,A -85,B 0,C 180,E1 10318.975,E2 10318.975} C_VEL
LIN {X 0,Y 410.186,Z 1241.392,A -85,B 0,C 180,E1 10323.508,E2 10323.508} C_VEL
LIN {X 0,Y 406.408,Z 1266.382,A -85,B 0,C 180,E1 10328.489,E2 10328.489} C_VEL
LIN {X 0,Y 404.111,Z 1285.868,A -85,B 0,C 180,E1 10333.735,E2 10333.735} C_VEL
LIN {X 0,Y 404.079,Z 1286.233,A -85,B 0,C 180,E1 10333.854,E2 10333.854} C_VEL
LIN {X 0,Y 401.201,Z 1291.073,A -85,B 0,C 180,E1 10335.545,E2 10335.545} C_VEL
LIN {X 0,Y 395.494,Z 1296.953,A -85,B 0,C 180,E1 10338.153,E2 10338.153} C_VEL
LIN {X 0,Y 395.36,Z 1297.558,A -85,B 0,C 180,E1 10338.46,E2 10338.46} C_VEL
LIN {X 0,Y 395.029,Z 1305.662,A -85,B 0,C 180,E1 10343.419,E2 10343.419} C_VEL
LIN {X 0,Y 394.928,Z 1309.193,A -85,B 0,C 180,E1 10347.809,E2 10347.809} C_VEL
LIN {X 0,Y 394.963,Z 1309.201,A -85,B 0,C 180,E1 10352.189,E2 10352.189} C_VEL
LIN {X 0,Y 395.004,Z 1304.43,A -85,B 0,C 180,E1 10357.573,E2 10357.573} C_VEL
LIN {X 0,Y 395.614,Z 1293.712,A -85,B 0,C 180,E1 10363.229,E2 10363.229} C_VEL
LIN {X 0,Y 397.211,Z 1276.598,A -85,B 0,C 180,E1 10368.972,E2 10368.972} C_VEL
LIN {X 0,Y 400.444,Z 1253.34,A -85,B 0,C 180,E1 10374.488,E2 10374.488} C_VEL
LIN {X 0,Y 405.179,Z 1226.325,A -85,B 0,C 180,E1 10379.262,E2 10379.262} C_VEL
LIN {X 0,Y 411.291,Z 1193.656,A -85,B 0,C 180,E1 10383.603,E2 10383.603} C_VEL
LIN {X 0,Y 417.751,Z 1159.212,A -85,B 0,C 180,E1 10386.997,E2 10386.997} C_VEL
LIN {X 0,Y 423.938,Z 1122.788,A -85,B 0,C 180,E1 10389.595,E2 10389.595} C_VEL
LIN {X 0,Y 429.283,Z 1084.65,A -85,B 0,C 180,E1 10391.435,E2 10391.435} C_VEL
LIN {X 0,Y 431.168,Z 1060.356,A -85,B 0,C 180,E1 10392.293,E2 10392.293} C_VEL
LIN {X 0,Y 413.96,Z 1025.361,A -85,B 0,C 180,E1 10395.437,E2 10395.437} C_VEL
LIN {X 0,Y 395.393,Z 994.581,A -85,B 0,C 180,E1 10398.924,E2 10398.924} C_VEL
LIN {X 0,Y 393.084,Z 989.03,A -85,B 0,C 180,E1 10399.504,E2 10399.504} C_VEL
LIN {X 0,Y 393.08,Z 989.03,A -85,B 0,C 180,E1 10404.843,E2 10404.843} C_VEL
LIN {X 0,Y 393.21,Z 989.03,A -85,B 0,C 180,E1 10411.964,E2 10411.964} C_VEL
LIN {X 0,Y 393.466,Z 989.03,A -85,B 0,C 180,E1 10417.449,E2 10417.449} C_VEL
LIN {X 0,Y 393.66,Z 989.03,A -85,B 0,C 180,E1 10424.436,E2 10424.436} C_VEL
LIN {X 0,Y 393.962,Z 989.03,A -85,B 0,C 180,E1 10431.187,E2 10431.187} C_VEL
LIN {X 0,Y 394.476,Z 989.03,A -85,B 0,C 180,E1 10437.808,E2 10437.808} C_VEL
LIN {X 0,Y 394.268,Z 989.03,A -85,B 0,C 180,E1 10444.39,E2 10444.39} C_VEL
LIN {X 0,Y 393.966,Z 989.03,A -85,B 0,C 180,E1 10451.041,E2 10451.041} C_VEL
LIN {X 0,Y 393.658,Z 989.03,A -85,B 0,C 180,E1 10457.857,E2 10457.857} C_VEL
LIN {X 0,Y 393.386,Z 989.03,A -85,B 0,C 180,E1 10464.957,E2 10464.957} C_VEL
LIN {X 0,Y 393.132,Z 989.03,A -85,B 0,C 180,E1 10472.504,E2 10472.504} C_VEL
LIN {X 0,Y 392.995,Z 989.03,A -85,B 0,C 180,E1 10479.831,E2 10479.831} C_VEL
LIN {X 0,Y 393.092,Z 989.662,A -85,B 0,C 180,E1 10484.365,E2 10484.365} C_VEL
LIN {X 0,Y 406.546,Z 1018.76,A -85,B 0,C 180,E1 10488.981,E2 10488.981} C_VEL
LIN {X 0,Y 415.668,Z 1046.781,A -85,B 0,C 180,E1 10493.314,E2 10493.314} C_VEL
LIN {X 0,Y 417.613,Z 1062.56,A -85,B 0,C 180,E1 10495.638,E2 10495.638} C_VEL
LIN {X 0,Y 411.042,Z 1091.921,A -85,B 0,C 180,E1 10499.537,E2 10499.537} C_VEL
LIN {X 0,Y 404.773,Z 1118.231,A -85,B 0,C 180,E1 10504.318,E2 10504.318} C_VEL
LIN {X 0,Y 400.022,Z 1138.939,A -85,B 0,C 180,E1 10509.578,E2 10509.578} C_VEL
LIN {X 0,Y 397.033,Z 1154.2,A -85,B 0,C 180,E1 10515.128,E2 10515.128} C_VEL
LIN {X 0,Y 395.749,Z 1163.316,A -85,B 0,C 180,E1 10520.121,E2 10520.121} C_VEL
LIN {X 0,Y 395.051,Z 1168.891,A -85,B 0,C 180,E1 10525.619,E2 10525.619} C_VEL
LIN {X 0,Y 395.124,Z 1170.234,A -85,B 0,C 180,E1 10530.001,E2 10530.001} C_VEL
LIN {X 0,Y 395.057,Z 1168.824,A -85,B 0,C 180,E1 10534.382,E2 10534.382} C_VEL
LIN {X 0,Y 395.713,Z 1163.179,A -85,B 0,C 180,E1 10539.882,E2 10539.882} C_VEL
LIN {X 0,Y 397.277,Z 1152.772,A -85,B 0,C 180,E1 10545.42,E2 10545.42} C_VEL
LIN {X 0,Y 400.439,Z 1136.766,A -85,B 0,C 180,E1 10550.978,E2 10550.978} C_VEL
LIN {X 0,Y 405.486,Z 1115.12,A -85,B 0,C 180,E1 10556.228,E2 10556.228} C_VEL
LIN {X 0,Y 411.506,Z 1089.851,A -85,B 0,C 180,E1 10560.682,E2 10560.682} C_VEL
LIN {X 0,Y 417.863,Z 1059.938,A -85,B 0,C 180,E1 10564.596,E2 10564.596} C_VEL
LIN {X 0,Y 413.63,Z 1039.542,A -85,B 0,C 180,E1 10567.712,E2 10567.712} C_VEL
LIN {X 0,Y 404.304,Z 1013.924,A -85,B 0,C 180,E1 10571.717,E2 10571.717} C_VEL
LIN {X 0,Y 393.1,Z 989.742,A -85,B 0,C 180,E1 10575.524,E2 10575.524} C_VEL
LIN {X 0,Y 393.141,Z 989.03,A -85,B 0,C 180,E1 10582.113,E2 10582.113} C_VEL
LIN {X 0,Y 393.215,Z 989.03,A -85,B 0,C 180,E1 10590.075,E2 10590.075} C_VEL
LIN {X 0,Y 393.477,Z 989.03,A -85,B 0,C 180,E1 10597.45,E2 10597.45} C_VEL
LIN {X 0,Y 393.673,Z 989.03,A -85,B 0,C 180,E1 10604.436,E2 10604.436} C_VEL
LIN {X 0,Y 394.029,Z 989.03,A -85,B 0,C 180,E1 10611.189,E2 10611.189} C_VEL
LIN {X 0,Y 394.488,Z 989.03,A -85,B 0,C 180,E1 10617.808,E2 10617.808} C_VEL
LIN {X 0,Y 394.284,Z 989.03,A -85,B 0,C 180,E1 10624.39,E2 10624.39} C_VEL
LIN {X 0,Y 393.977,Z 989.03,A -85,B 0,C 180,E1 10631.04,E2 10631.04} C_VEL
LIN {X 0,Y 393.656,Z 989.03,A -85,B 0,C 180,E1 10637.858,E2 10637.858} C_VEL
LIN {X 0,Y 393.395,Z 989.03,A -85,B 0,C 180,E1 10644.956,E2 10644.956} C_VEL
LIN {X 0,Y 393.241,Z 989.03,A -85,B 0,C 180,E1 10652.494,E2 10652.494} C_VEL
LIN {X 0,Y 393.112,Z 989.03,A -85,B 0,C 180,E1 10659.849,E2 10659.849} C_VEL
LIN {X 0,Y 393.051,Z 989.03,A -85,B 0,C 180,E1 10660.559,E2 10660.559} C_VEL
LIN {X 0,Y 395.327,Z 994.568,A -85,B 0,C 180,E1 10661.079,E2 10661.079} C_VEL
LIN {X 0,Y 415.684,Z 1028.542,A -85,B 0,C 180,E1 10664.877,E2 10664.877} C_VEL
LIN {X 0,Y 431.568,Z 1060.964,A -85,B 0,C 180,E1 10667.776,E2 10667.776} C_VEL
LIN {X 0,Y 426.831,Z 1103.358,A -85,B 0,C 180,E1 10669.363,E2 10669.363} C_VEL
LIN {X 0,Y 420.91,Z 1141.584,A -85,B 0,C 180,E1 10671.634,E2 10671.634} C_VEL
LIN {X 0,Y 414.428,Z 1177.378,A -85,B 0,C 180,E1 10674.663,E2 10674.663} C_VEL
LIN {X 0,Y 407.899,Z 1211.628,A -85,B 0,C 180,E1 10678.628,E2 10678.628} C_VEL
LIN {X 0,Y 402.478,Z 1241.49,A -85,B 0,C 180,E1 10683.261,E2 10683.261} C_VEL
LIN {X 0,Y 398.585,Z 1266.118,A -85,B 0,C 180,E1 10688.339,E2 10688.339} C_VEL
LIN {X 0,Y 396.306,Z 1284.433,A -85,B 0,C 180,E1 10693.406,E2 10693.406} C_VEL
LIN {X 0,Y 395.36,Z 1297.558,A -85,B 0,C 180,E1 10698.46,E2 10698.46} C_VEL
LIN {X 0,Y 392.729,Z 1300.74,A -85,B 0,C 180,E1 10700.274,E2 10700.274} C_VEL
LIN {X 0,Y 387.197,Z 1304.359,A -85,B 0,C 180,E1 10703.366,E2 10703.366} C_VEL
LIN {X 0,Y 387.134,Z 1307.817,A -85,B 0,C 180,E1 10707.765,E2 10707.765} C_VEL
LIN {X 0,Y 387.167,Z 1307.824,A -85,B 0,C 180,E1 10712.233,E2 10712.233} C_VEL
LIN {X 0,Y 387.19,Z 1302.899,A -85,B 0,C 180,E1 10717.839,E2 10717.839} C_VEL
LIN {X 0,Y 387.807,Z 1292.296,A -85,B 0,C 180,E1 10723.501,E2 10723.501} C_VEL
LIN {X 0,Y 389.415,Z 1275.598,A -85,B 0,C 180,E1 10729.23,E2 10729.23} C_VEL
